   1:L PR[91] R[100]mm/sec CNT100;
   1:  PR[GP1:91,1] = PR[GP1:90,1] + 70.472;
   1:  PR[GP1:91,2] = PR[GP1:90,2] + 15.297;
   1:L PR[91] R[100]mm/sec CNT100;
   1:  PR[GP1:91,1] = PR[GP1:90,1] + 68.185;
   1:  PR[GP1:91,2] = PR[GP1:90,2] + 19.487;
   1:L PR[91] R[100]mm/sec CNT100;
   1:  PR[GP1:91,1] = PR[GP1:90,1] + 65.966;
   1:  PR[GP1:91,2] = PR[GP1:90,2] + 22.379;
   1:L PR[91] R[100]mm/sec CNT100;
   1:  PR[GP1:91,1] = PR[GP1:90,1] + 63.212;
   1:  PR[GP1:91,2] = PR[GP1:90,2] + 24.842;
   1:L PR[91] R[100]mm/sec CNT100;
   1:  PR[GP1:91,1] = PR[GP1:90,1] + 59.563;
   1:  PR[GP1:91,2] = PR[GP1:90,2] + 28.170;
   1:L PR[91] R[100]mm/sec CNT100;
   1:  PR[GP1:91,1] = PR[GP1:90,1] + 56.581;
   1:  PR[GP1:91,2] = PR[GP1:90,2] + 29.968;
   1:L PR[91] R[100]mm/sec CNT100;
   1:  PR[GP1:91,1] = PR[GP1:90,1] + 53.246;
   1:  PR[GP1:91,2] = PR[GP1:90,2] + 31.207;
   1:L PR[91] R[100]mm/sec CNT100;
   1:  PR[GP1:91,1] = PR[GP1:90,1] + 48.490;
   1:  PR[GP1:91,2] = PR[GP1:90,2] + 33.267;
   1:L PR[91] R[100]mm/sec CNT100;
   1:  PR[GP1:91,1] = PR[GP1:90,1] + 45.251;
   1:  PR[GP1:91,2] = PR[GP1:90,2] + 33.819;
   1:L PR[91] R[100]mm/sec CNT100;
   1:  PR[GP1:91,1] = PR[GP1:90,1] + 39.491;
   1:  PR[GP1:91,2] = PR[GP1:90,2] + 34.252;
   1:L PR[91] R[100]mm/sec CNT100;
   1:  PR[GP1:91,1] = PR[GP1:90,1] + 36.457;
   1:  PR[GP1:91,2] = PR[GP1:90,2] + 34.197;
   1:L PR[91] R[100]mm/sec CNT100;
   1:  PR[GP1:91,1] = PR[GP1:90,1] + 33.474;
   1:  PR[GP1:91,2] = PR[GP1:90,2] + 33.576;
   1:L PR[91] R[100]mm/sec CNT100;
   1:  PR[GP1:91,1] = PR[GP1:90,1] + 27.456;
   1:  PR[GP1:91,2] = PR[GP1:90,2] + 32.002;
   1:L PR[91] R[100]mm/sec CNT100;
   1:  PR[GP1:91,1] = PR[GP1:90,1] + 24.948;
   1:  PR[GP1:91,2] = PR[GP1:90,2] + 30.965;
   1:L PR[91] R[100]mm/sec CNT100;
   1:  PR[GP1:91,1] = PR[GP1:90,1] + 22.645;
   1:  PR[GP1:91,2] = PR[GP1:90,2] + 29.460;
   1:L PR[91] R[100]mm/sec CNT100;
   1:  PR[GP1:91,1] = PR[GP1:90,1] + 17.064;
   1:  PR[GP1:91,2] = PR[GP1:90,2] + 25.755;
   1:L PR[91] R[100]mm/sec CNT100;
   1:  PR[GP1:91,1] = PR[GP1:90,1] + 15.344;
   1:  PR[GP1:91,2] = PR[GP1:90,2] + 24.100;
   1:L PR[91] R[100]mm/sec CNT100;
   1:  PR[GP1:91,1] = PR[GP1:90,1] + 13.923;
   1:  PR[GP1:91,2] = PR[GP1:90,2] + 22.102;
   1:L PR[91] R[100]mm/sec CNT100;
   1:  PR[GP1:91,1] = PR[GP1:90,1] + 9.561;
   1:  PR[GP1:91,2] = PR[GP1:90,2] + 16.404;
   1:L PR[91] R[100]mm/sec CNT100;
   1:  PR[GP1:91,1] = PR[GP1:90,1] + 8.670;
   1:  PR[GP1:91,2] = PR[GP1:90,2] + 14.466;
   1:L PR[91] R[100]mm/sec CNT100;
   1:  PR[GP1:91,1] = PR[GP1:90,1] + 6.222;
   1:  PR[GP1:91,2] = PR[GP1:90,2] + 7.080;
   1:L PR[91] R[100]mm/sec CNT100;
   1:  PR[GP1:91,1] = PR[GP1:90,1] + 5.845;
   1:  PR[GP1:91,2] = PR[GP1:90,2] + 5.563;
   1:L PR[91] R[100]mm/sec CNT100;
   1:  PR[GP1:91,1] = PR[GP1:90,1] + 5.869;
   1:  PR[GP1:91,2] = PR[GP1:90,2] + 5.549;
   1:L PR[91] R[100]mm/sec CNT100;
   1:  PR[GP1:91,1] = PR[GP1:90,1] + 5.812;
   1:  PR[GP1:91,2] = PR[GP1:90,2] + 5.029;
   1:L PR[91] R[100]mm/sec CNT100;
   1:  PR[GP1:91,1] = PR[GP1:90,1] + 5.410;
   1:  PR[GP1:91,2] = PR[GP1:90,2] + 4.073;
   1:L PR[91] R[100]mm/sec CNT100;
   1:  PR[GP1:91,1] = PR[GP1:90,1] + 5.006;
   1:  PR[GP1:91,2] = PR[GP1:90,2] + 3.295;
   1:L PR[91] R[100]mm/sec CNT100;
   1:  PR[GP1:91,1] = PR[GP1:90,1] + 4.488;
   1:  PR[GP1:91,2] = PR[GP1:90,2] + 2.358;
   1:L PR[91] R[100]mm/sec CNT100;
   1:  PR[GP1:91,1] = PR[GP1:90,1] + 3.900;
   1:  PR[GP1:91,2] = PR[GP1:90,2] + 1.720;
   1:L PR[91] R[100]mm/sec CNT100;
   1:  PR[GP1:91,1] = PR[GP1:90,1] + 3.010;
   1:  PR[GP1:91,2] = PR[GP1:90,2] + 1.107;
   1:L PR[91] R[100]mm/sec CNT100;
   1:  PR[GP1:91,1] = PR[GP1:90,1] + 2.104;
   1:  PR[GP1:91,2] = PR[GP1:90,2] + 0.771;
   1:L PR[91] R[100]mm/sec CNT100;
   1:  PR[GP1:91,1] = PR[GP1:90,1] + 1.542;
   1:  PR[GP1:91,2] = PR[GP1:90,2] + 0.621;
   1:L PR[91] R[100]mm/sec CNT100;
   1:  PR[GP1:91,1] = PR[GP1:90,1] + 0.324;
   1:  PR[GP1:91,2] = PR[GP1:90,2] + 0.328;
   1:L PR[91] R[100]mm/sec CNT100;
   1:  PR[GP1:91,1] = PR[GP1:90,1] + -0.154;
   1:L PR[91] R[100]mm/sec CNT100;
   1:  ! -- Layer/Ebene 22 -- !;
   1:  PR[91] = PR[90];
   1:  PR[GP1:91,1] = PR[GP1:90,1] + -0.443;
   1:  PR[GP1:91,2] = PR[GP1:90,2] + 0.471;
   1:  PR[GP1:91,3] = PR[GP1:90,3] + 13.725;
   1:L PR[91] R[100]mm/sec CNT100;
   1:  PR[GP1:91,1] = PR[GP1:90,1] + -0.647;
   1:  PR[GP1:91,2] = PR[GP1:90,2] + 0.480;
   1:L PR[91] R[100]mm/sec CNT100;
   1:  PR[GP1:91,1] = PR[GP1:90,1] + -3.627;
   1:  PR[GP1:91,2] = PR[GP1:90,2] + 1.659;
   1:L PR[91] R[100]mm/sec CNT100;
   1:  PR[GP1:91,1] = PR[GP1:90,1] + -3.980;
   1:  PR[GP1:91,2] = PR[GP1:90,2] + 2.296;
   1:L PR[91] R[100]mm/sec CNT100;
   1:  PR[GP1:91,1] = PR[GP1:90,1] + -4.040;
   1:  PR[GP1:91,2] = PR[GP1:90,2] + 2.351;
   1:L PR[91] R[100]mm/sec CNT100;
   1:  PR[GP1:91,1] = PR[GP1:90,1] + -4.473;
   1:  PR[GP1:91,2] = PR[GP1:90,2] + 3.055;
   1:L PR[91] R[100]mm/sec CNT100;
   1:  PR[GP1:91,1] = PR[GP1:90,1] + -5.526;
   1:  PR[GP1:91,2] = PR[GP1:90,2] + 4.999;
   1:L PR[91] R[100]mm/sec CNT100;
   1:  PR[GP1:91,1] = PR[GP1:90,1] + -5.589;
   1:  PR[GP1:91,2] = PR[GP1:90,2] + 5.579;
   1:L PR[91] R[100]mm/sec CNT100;
   1:  PR[GP1:91,1] = PR[GP1:90,1] + -5.827;
   1:  PR[GP1:91,2] = PR[GP1:90,2] + 6.538;
   1:L PR[91] R[100]mm/sec CNT100;
   1:  PR[GP1:91,1] = PR[GP1:90,1] + -8.589;
   1:  PR[GP1:91,2] = PR[GP1:90,2] + 14.871;
   1:L PR[91] R[100]mm/sec CNT100;
   1:  PR[GP1:91,1] = PR[GP1:90,1] + -9.257;
   1:  PR[GP1:91,2] = PR[GP1:90,2] + 16.324;
   1:L PR[91] R[100]mm/sec CNT100;
   1:  PR[GP1:91,1] = PR[GP1:90,1] + -10.196;
   1:  PR[GP1:91,2] = PR[GP1:90,2] + 17.645;
   1:L PR[91] R[100]mm/sec CNT100;
   1:  PR[GP1:91,1] = PR[GP1:90,1] + -15.288;
   1:  PR[GP1:91,2] = PR[GP1:90,2] + 24.311;
   1:L PR[91] R[100]mm/sec CNT100;
   1:  PR[GP1:91,1] = PR[GP1:90,1] + -16.646;
   1:  PR[GP1:91,2] = PR[GP1:90,2] + 25.617;
   1:L PR[91] R[100]mm/sec CNT100;
   1:  PR[GP1:91,1] = PR[GP1:90,1] + -18.262;
   1:  PR[GP1:91,2] = PR[GP1:90,2] + 26.674;
   1:L PR[91] R[100]mm/sec CNT100;
   1:  PR[GP1:91,1] = PR[GP1:90,1] + -24.852;
   1:  PR[GP1:91,2] = PR[GP1:90,2] + 31.045;
   1:L PR[91] R[100]mm/sec CNT100;
   1:  PR[GP1:91,1] = PR[GP1:90,1] + -26.907;
   1:  PR[GP1:91,2] = PR[GP1:90,2] + 31.895;
   1:L PR[91] R[100]mm/sec CNT100;
   1:  PR[GP1:91,1] = PR[GP1:90,1] + -29.156;
   1:  PR[GP1:91,2] = PR[GP1:90,2] + 32.362;
   1:L PR[91] R[100]mm/sec CNT100;
   1:  PR[GP1:91,1] = PR[GP1:90,1] + -36.283;
   1:  PR[GP1:91,2] = PR[GP1:90,2] + 34.208;
   1:L PR[91] R[100]mm/sec CNT100;
   1:  PR[GP1:91,1] = PR[GP1:90,1] + -38.869;
   1:  PR[GP1:91,2] = PR[GP1:90,2] + 34.255;
   1:L PR[91] R[100]mm/sec CNT100;
   1:  PR[GP1:91,1] = PR[GP1:90,1] + -45.366;
   1:  PR[GP1:91,2] = PR[GP1:90,2] + 33.766;
   1:L PR[91] R[100]mm/sec CNT100;
   1:  PR[GP1:91,1] = PR[GP1:90,1] + -48.228;
   1:  PR[GP1:91,2] = PR[GP1:90,2] + 33.279;
   1:L PR[91] R[100]mm/sec CNT100;
   1:  PR[GP1:91,1] = PR[GP1:90,1] + -50.961;
   1:  PR[GP1:91,2] = PR[GP1:90,2] + 32.263;
   1:L PR[91] R[100]mm/sec CNT100;
   1:  PR[GP1:91,1] = PR[GP1:90,1] + -56.550;
   1:  PR[GP1:91,2] = PR[GP1:90,2] + 29.856;
   1:L PR[91] R[100]mm/sec CNT100;
   1:  PR[GP1:91,1] = PR[GP1:90,1] + -59.229;
   1:  PR[GP1:91,2] = PR[GP1:90,2] + 28.240;
   1:L PR[91] R[100]mm/sec CNT100;
   1:  PR[GP1:91,1] = PR[GP1:90,1] + -61.590;
   1:  PR[GP1:91,2] = PR[GP1:90,2] + 26.129;
   1:L PR[91] R[100]mm/sec CNT100;
   1:  PR[GP1:91,1] = PR[GP1:90,1] + -65.832;
   1:  PR[GP1:91,2] = PR[GP1:90,2] + 22.263;
   1:L PR[91] R[100]mm/sec CNT100;
   1:  PR[GP1:91,1] = PR[GP1:90,1] + -67.832;
   1:  PR[GP1:91,2] = PR[GP1:90,2] + 19.657;
   1:L PR[91] R[100]mm/sec CNT100;
   1:  PR[GP1:91,1] = PR[GP1:90,1] + -69.340;
   1:  PR[GP1:91,2] = PR[GP1:90,2] + 16.667;
   1:L PR[91] R[100]mm/sec CNT100;
   1:  PR[GP1:91,1] = PR[GP1:90,1] + -71.966;
   1:  PR[GP1:91,2] = PR[GP1:90,2] + 11.848;
   1:L PR[91] R[100]mm/sec CNT100;
   1:  PR[GP1:91,1] = PR[GP1:90,1] + -72.899;
   1:  PR[GP1:91,2] = PR[GP1:90,2] + 8.606;
   1:L PR[91] R[100]mm/sec CNT100;
   1:  PR[GP1:91,1] = PR[GP1:90,1] + -73.222;
   1:  PR[GP1:91,2] = PR[GP1:90,2] + 5.161;
   1:L PR[91] R[100]mm/sec CNT100;
   1:  PR[GP1:91,1] = PR[GP1:90,1] + -74.099;
   1:  PR[GP1:91,2] = PR[GP1:90,2] + -0.094;
   1:L PR[91] R[100]mm/sec CNT100;
   1:  PR[GP1:91,1] = PR[GP1:90,1] + -73.772;
   1:  PR[GP1:91,2] = PR[GP1:90,2] + -3.582;
   1:L PR[91] R[100]mm/sec CNT100;
   1:  PR[GP1:91,1] = PR[GP1:90,1] + -72.906;
   1:  PR[GP1:91,2] = PR[GP1:90,2] + -8.729;
   1:L PR[91] R[100]mm/sec CNT100;
   1:  PR[GP1:91,1] = PR[GP1:90,1] + -71.963;
   1:  PR[GP1:91,2] = PR[GP1:90,2] + -12.001;
   1:L PR[91] R[100]mm/sec CNT100;
   1:  PR[GP1:91,1] = PR[GP1:90,1] + -70.418;
   1:  PR[GP1:91,2] = PR[GP1:90,2] + -15.062;
   1:L PR[91] R[100]mm/sec CNT100;
   1:  PR[GP1:91,1] = PR[GP1:90,1] + -67.838;
   1:  PR[GP1:91,2] = PR[GP1:90,2] + -19.793;
   1:L PR[91] R[100]mm/sec CNT100;
   1:  PR[GP1:91,1] = PR[GP1:90,1] + -65.834;
   1:  PR[GP1:91,2] = PR[GP1:90,2] + -22.405;
   1:L PR[91] R[100]mm/sec CNT100;
   1:  PR[GP1:91,1] = PR[GP1:90,1] + -63.343;
   1:  PR[GP1:91,2] = PR[GP1:90,2] + -24.632;
   1:L PR[91] R[100]mm/sec CNT100;
   1:  PR[GP1:91,1] = PR[GP1:90,1] + -59.227;
   1:  PR[GP1:91,2] = PR[GP1:90,2] + -28.385;
   1:L PR[91] R[100]mm/sec CNT100;
   1:  PR[GP1:91,1] = PR[GP1:90,1] + -56.563;
   1:  PR[GP1:91,2] = PR[GP1:90,2] + -29.992;
   1:L PR[91] R[100]mm/sec CNT100;
   1:  PR[GP1:91,1] = PR[GP1:90,1] + -53.577;
   1:  PR[GP1:91,2] = PR[GP1:90,2] + -31.101;
   1:L PR[91] R[100]mm/sec CNT100;
   1:  PR[GP1:91,1] = PR[GP1:90,1] + -48.212;
   1:  PR[GP1:91,2] = PR[GP1:90,2] + -33.425;
   1:L PR[91] R[100]mm/sec CNT100;
   1:  PR[GP1:91,1] = PR[GP1:90,1] + -45.366;
   1:  PR[GP1:91,2] = PR[GP1:90,2] + -33.910;
   1:L PR[91] R[100]mm/sec CNT100;
   1:  PR[GP1:91,1] = PR[GP1:90,1] + -38.869;
   1:  PR[GP1:91,2] = PR[GP1:90,2] + -34.399;
   1:L PR[91] R[100]mm/sec CNT100;
   1:  PR[GP1:91,1] = PR[GP1:90,1] + -36.268;
   1:  PR[GP1:91,2] = PR[GP1:90,2] + -34.352;
   1:L PR[91] R[100]mm/sec CNT100;
   1:  PR[GP1:91,1] = PR[GP1:90,1] + -33.709;
   1:  PR[GP1:91,2] = PR[GP1:90,2] + -33.819;
   1:L PR[91] R[100]mm/sec CNT100;
   1:  PR[GP1:91,1] = PR[GP1:90,1] + -26.921;
   1:  PR[GP1:91,2] = PR[GP1:90,2] + -32.044;
   1:L PR[91] R[100]mm/sec CNT100;
   1:  PR[GP1:91,1] = PR[GP1:90,1] + -24.850;
   1:  PR[GP1:91,2] = PR[GP1:90,2] + -31.188;
   1:L PR[91] R[100]mm/sec CNT100;
   1:  PR[GP1:91,1] = PR[GP1:90,1] + -22.942;
   1:  PR[GP1:91,2] = PR[GP1:90,2] + -29.941;
   1:L PR[91] R[100]mm/sec CNT100;
   1:  PR[GP1:91,1] = PR[GP1:90,1] + -16.647;
   1:  PR[GP1:91,2] = PR[GP1:90,2] + -25.762;
   1:L PR[91] R[100]mm/sec CNT100;
   1:  PR[GP1:91,1] = PR[GP1:90,1] + -15.296;
   1:  PR[GP1:91,2] = PR[GP1:90,2] + -24.463;
   1:L PR[91] R[100]mm/sec CNT100;
   1:  PR[GP1:91,1] = PR[GP1:90,1] + -14.172;
   1:  PR[GP1:91,2] = PR[GP1:90,2] + -22.882;
   1:L PR[91] R[100]mm/sec CNT100;
   1:  PR[GP1:91,1] = PR[GP1:90,1] + -9.252;
   1:  PR[GP1:91,2] = PR[GP1:90,2] + -16.458;
   1:L PR[91] R[100]mm/sec CNT100;
   1:  PR[GP1:91,1] = PR[GP1:90,1] + -8.589;
   1:  PR[GP1:91,2] = PR[GP1:90,2] + -15.015;
   1:L PR[91] R[100]mm/sec CNT100;
   1:  PR[GP1:91,1] = PR[GP1:90,1] + -5.828;
   1:  PR[GP1:91,2] = PR[GP1:90,2] + -6.684;
   1:L PR[91] R[100]mm/sec CNT100;
   1:  PR[GP1:91,1] = PR[GP1:90,1] + -5.587;
   1:  PR[GP1:91,2] = PR[GP1:90,2] + -5.718;
   1:L PR[91] R[100]mm/sec CNT100;
   1:  PR[GP1:91,1] = PR[GP1:90,1] + -5.590;
   1:  PR[GP1:91,2] = PR[GP1:90,2] + -5.716;
   1:L PR[91] R[100]mm/sec CNT100;
   1:  PR[GP1:91,1] = PR[GP1:90,1] + -5.530;
   1:  PR[GP1:91,2] = PR[GP1:90,2] + -5.173;
   1:L PR[91] R[100]mm/sec CNT100;
   1:  PR[GP1:91,1] = PR[GP1:90,1] + -4.941;
   1:  PR[GP1:91,2] = PR[GP1:90,2] + -3.769;
   1:L PR[91] R[100]mm/sec CNT100;
   1:  PR[GP1:91,1] = PR[GP1:90,1] + -4.300;
   1:  PR[GP1:91,2] = PR[GP1:90,2] + -2.578;
   1:L PR[91] R[100]mm/sec CNT100;
   1:  PR[GP1:91,1] = PR[GP1:90,1] + -3.647;
   1:  PR[GP1:91,2] = PR[GP1:90,2] + -1.869;
   1:L PR[91] R[100]mm/sec CNT100;
   1:  PR[GP1:91,1] = PR[GP1:90,1] + -2.659;
   1:  PR[GP1:91,2] = PR[GP1:90,2] + -1.188;
   1:L PR[91] R[100]mm/sec CNT100;
   1:  PR[GP1:91,1] = PR[GP1:90,1] + -2.064;
   1:  PR[GP1:91,2] = PR[GP1:90,2] + -0.967;
   1:L PR[91] R[100]mm/sec CNT100;
   1:  PR[GP1:91,1] = PR[GP1:90,1] + -1.705;
   1:  PR[GP1:91,2] = PR[GP1:90,2] + -0.872;
   1:L PR[91] R[100]mm/sec CNT100;
   1:  PR[GP1:91,1] = PR[GP1:90,1] + -0.043;
   1:  PR[GP1:91,2] = PR[GP1:90,2] + -0.472;
   1:L PR[91] R[100]mm/sec CNT100;
   1:  PR[GP1:91,1] = PR[GP1:90,1] + 0.299;
   1:L PR[91] R[100]mm/sec CNT100;
   1:  PR[GP1:91,1] = PR[GP1:90,1] + 0.657;
   1:  PR[GP1:91,2] = PR[GP1:90,2] + -0.615;
   1:L PR[91] R[100]mm/sec CNT100;
   1:  PR[GP1:91,1] = PR[GP1:90,1] + 0.860;
   1:  PR[GP1:91,2] = PR[GP1:90,2] + -0.623;
   1:L PR[91] R[100]mm/sec CNT100;
   1:  PR[GP1:91,1] = PR[GP1:90,1] + 3.841;
   1:  PR[GP1:91,2] = PR[GP1:90,2] + -1.803;
   1:L PR[91] R[100]mm/sec CNT100;
   1:  PR[GP1:91,1] = PR[GP1:90,1] + 4.193;
   1:  PR[GP1:91,2] = PR[GP1:90,2] + -2.440;
   1:L PR[91] R[100]mm/sec CNT100;
   1:  PR[GP1:91,1] = PR[GP1:90,1] + 4.254;
   1:  PR[GP1:91,2] = PR[GP1:90,2] + -2.495;
   1:L PR[91] R[100]mm/sec CNT100;
   1:  PR[GP1:91,1] = PR[GP1:90,1] + 4.687;
   1:  PR[GP1:91,2] = PR[GP1:90,2] + -3.199;
   1:L PR[91] R[100]mm/sec CNT100;
   1:  PR[GP1:91,1] = PR[GP1:90,1] + 5.739;
   1:  PR[GP1:91,2] = PR[GP1:90,2] + -5.143;
   1:L PR[91] R[100]mm/sec CNT100;
   1:  PR[GP1:91,1] = PR[GP1:90,1] + 5.802;
   1:  PR[GP1:91,2] = PR[GP1:90,2] + -5.723;
   1:L PR[91] R[100]mm/sec CNT100;
   1:  PR[GP1:91,1] = PR[GP1:90,1] + 6.040;
   1:  PR[GP1:91,2] = PR[GP1:90,2] + -6.685;
   1:L PR[91] R[100]mm/sec CNT100;
   1:  PR[GP1:91,1] = PR[GP1:90,1] + 8.801;
   1:  PR[GP1:91,2] = PR[GP1:90,2] + -15.012;
   1:L PR[91] R[100]mm/sec CNT100;
   1:  PR[GP1:91,1] = PR[GP1:90,1] + 9.469;
   1:  PR[GP1:91,2] = PR[GP1:90,2] + -16.464;
   1:L PR[91] R[100]mm/sec CNT100;
   1:  PR[GP1:91,1] = PR[GP1:90,1] + 10.408;
   1:  PR[GP1:91,2] = PR[GP1:90,2] + -17.786;
   1:L PR[91] R[100]mm/sec CNT100;
   1:  PR[GP1:91,1] = PR[GP1:90,1] + 15.500;
   1:  PR[GP1:91,2] = PR[GP1:90,2] + -24.455;
   1:L PR[91] R[100]mm/sec CNT100;
   1:  PR[GP1:91,1] = PR[GP1:90,1] + 16.857;
   1:  PR[GP1:91,2] = PR[GP1:90,2] + -25.760;
   1:L PR[91] R[100]mm/sec CNT100;
   1:  PR[GP1:91,1] = PR[GP1:90,1] + 18.474;
   1:  PR[GP1:91,2] = PR[GP1:90,2] + -26.817;
   1:L PR[91] R[100]mm/sec CNT100;
   1:  PR[GP1:91,1] = PR[GP1:90,1] + 25.063;
   1:  PR[GP1:91,2] = PR[GP1:90,2] + -31.188;
   1:L PR[91] R[100]mm/sec CNT100;
   1:  PR[GP1:91,1] = PR[GP1:90,1] + 27.119;
   1:  PR[GP1:91,2] = PR[GP1:90,2] + -32.038;
   1:L PR[91] R[100]mm/sec CNT100;
   1:  PR[GP1:91,1] = PR[GP1:90,1] + 29.367;
   1:  PR[GP1:91,2] = PR[GP1:90,2] + -32.506;
   1:L PR[91] R[100]mm/sec CNT100;
   1:  PR[GP1:91,1] = PR[GP1:90,1] + 36.495;
   1:  PR[GP1:91,2] = PR[GP1:90,2] + -34.352;
   1:L PR[91] R[100]mm/sec CNT100;
   1:  PR[GP1:91,1] = PR[GP1:90,1] + 39.081;
   1:  PR[GP1:91,2] = PR[GP1:90,2] + -34.399;
   1:L PR[91] R[100]mm/sec CNT100;
   1:  PR[GP1:91,1] = PR[GP1:90,1] + 45.579;
   1:  PR[GP1:91,2] = PR[GP1:90,2] + -33.910;
   1:L PR[91] R[100]mm/sec CNT100;
   1:  PR[GP1:91,1] = PR[GP1:90,1] + 48.441;
   1:  PR[GP1:91,2] = PR[GP1:90,2] + -33.423;
   1:L PR[91] R[100]mm/sec CNT100;
   1:  PR[GP1:91,1] = PR[GP1:90,1] + 51.174;
   1:  PR[GP1:91,2] = PR[GP1:90,2] + -32.407;
   1:L PR[91] R[100]mm/sec CNT100;
   1:  PR[GP1:91,1] = PR[GP1:90,1] + 56.763;
   1:  PR[GP1:91,2] = PR[GP1:90,2] + -30.000;
   1:L PR[91] R[100]mm/sec CNT100;
   1:  PR[GP1:91,1] = PR[GP1:90,1] + 59.442;
   1:  PR[GP1:91,2] = PR[GP1:90,2] + -28.385;
   1:L PR[91] R[100]mm/sec CNT100;
   1:  PR[GP1:91,1] = PR[GP1:90,1] + 61.803;
   1:  PR[GP1:91,2] = PR[GP1:90,2] + -26.274;
   1:L PR[91] R[100]mm/sec CNT100;
   1:  PR[GP1:91,1] = PR[GP1:90,1] + 66.045;
   1:  PR[GP1:91,2] = PR[GP1:90,2] + -22.407;
   1:L PR[91] R[100]mm/sec CNT100;
   1:  PR[GP1:91,1] = PR[GP1:90,1] + 68.045;
   1:  PR[GP1:91,2] = PR[GP1:90,2] + -19.800;
   1:L PR[91] R[100]mm/sec CNT100;
   1:  PR[GP1:91,1] = PR[GP1:90,1] + 69.553;
   1:  PR[GP1:91,2] = PR[GP1:90,2] + -16.810;
   1:L PR[91] R[100]mm/sec CNT100;
   1:  PR[GP1:91,1] = PR[GP1:90,1] + 72.179;
   1:  PR[GP1:91,2] = PR[GP1:90,2] + -11.994;
   1:L PR[91] R[100]mm/sec CNT100;
   1:  PR[GP1:91,1] = PR[GP1:90,1] + 73.113;
   1:  PR[GP1:91,2] = PR[GP1:90,2] + -8.752;
   1:L PR[91] R[100]mm/sec CNT100;
   1:  PR[GP1:91,1] = PR[GP1:90,1] + 73.436;
   1:  PR[GP1:91,2] = PR[GP1:90,2] + -5.307;
   1:L PR[91] R[100]mm/sec CNT100;
   1:  PR[GP1:91,1] = PR[GP1:90,1] + 74.312;
   1:  PR[GP1:91,2] = PR[GP1:90,2] + -0.050;
   1:L PR[91] R[100]mm/sec CNT100;
   1:  PR[GP1:91,1] = PR[GP1:90,1] + 73.985;
   1:  PR[GP1:91,2] = PR[GP1:90,2] + 3.438;
   1:L PR[91] R[100]mm/sec CNT100;
   1:  PR[GP1:91,1] = PR[GP1:90,1] + 73.119;
   1:  PR[GP1:91,2] = PR[GP1:90,2] + 8.587;
   1:L PR[91] R[100]mm/sec CNT100;
   1:  PR[GP1:91,1] = PR[GP1:90,1] + 72.176;
   1:  PR[GP1:91,2] = PR[GP1:90,2] + 11.859;
   1:L PR[91] R[100]mm/sec CNT100;
   1:  PR[GP1:91,1] = PR[GP1:90,1] + 70.632;
   1:  PR[GP1:91,2] = PR[GP1:90,2] + 14.920;
   1:L PR[91] R[100]mm/sec CNT100;
   1:  PR[GP1:91,1] = PR[GP1:90,1] + 68.051;
   1:  PR[GP1:91,2] = PR[GP1:90,2] + 19.648;
   1:L PR[91] R[100]mm/sec CNT100;
   1:  PR[GP1:91,1] = PR[GP1:90,1] + 66.047;
   1:  PR[GP1:91,2] = PR[GP1:90,2] + 22.260;
   1:L PR[91] R[100]mm/sec CNT100;
   1:  PR[GP1:91,1] = PR[GP1:90,1] + 63.556;
   1:  PR[GP1:91,2] = PR[GP1:90,2] + 24.488;
   1:L PR[91] R[100]mm/sec CNT100;
   1:  PR[GP1:91,1] = PR[GP1:90,1] + 59.439;
   1:  PR[GP1:91,2] = PR[GP1:90,2] + 28.242;
   1:L PR[91] R[100]mm/sec CNT100;
   1:  PR[GP1:91,1] = PR[GP1:90,1] + 56.776;
   1:  PR[GP1:91,2] = PR[GP1:90,2] + 29.848;
   1:L PR[91] R[100]mm/sec CNT100;
   1:  PR[GP1:91,1] = PR[GP1:90,1] + 53.790;
   1:  PR[GP1:91,2] = PR[GP1:90,2] + 30.958;
   1:L PR[91] R[100]mm/sec CNT100;
   1:  PR[GP1:91,1] = PR[GP1:90,1] + 48.425;
   1:  PR[GP1:91,2] = PR[GP1:90,2] + 33.281;
   1:L PR[91] R[100]mm/sec CNT100;
   1:  PR[GP1:91,1] = PR[GP1:90,1] + 45.579;
   1:  PR[GP1:91,2] = PR[GP1:90,2] + 33.766;
   1:L PR[91] R[100]mm/sec CNT100;
   1:  PR[GP1:91,1] = PR[GP1:90,1] + 39.081;
   1:  PR[GP1:91,2] = PR[GP1:90,2] + 34.255;
   1:L PR[91] R[100]mm/sec CNT100;
   1:  PR[GP1:91,1] = PR[GP1:90,1] + 36.480;
   1:  PR[GP1:91,2] = PR[GP1:90,2] + 34.208;
   1:L PR[91] R[100]mm/sec CNT100;
   1:  PR[GP1:91,1] = PR[GP1:90,1] + 33.921;
   1:  PR[GP1:91,2] = PR[GP1:90,2] + 33.675;
   1:L PR[91] R[100]mm/sec CNT100;
   1:  PR[GP1:91,1] = PR[GP1:90,1] + 27.133;
   1:  PR[GP1:91,2] = PR[GP1:90,2] + 31.900;
   1:L PR[91] R[100]mm/sec CNT100;
   1:  PR[GP1:91,1] = PR[GP1:90,1] + 25.062;
   1:  PR[GP1:91,2] = PR[GP1:90,2] + 31.043;
   1:L PR[91] R[100]mm/sec CNT100;
   1:  PR[GP1:91,1] = PR[GP1:90,1] + 23.153;
   1:  PR[GP1:91,2] = PR[GP1:90,2] + 29.796;
   1:L PR[91] R[100]mm/sec CNT100;
   1:  PR[GP1:91,1] = PR[GP1:90,1] + 16.859;
   1:  PR[GP1:91,2] = PR[GP1:90,2] + 25.618;
   1:L PR[91] R[100]mm/sec CNT100;
   1:  PR[GP1:91,1] = PR[GP1:90,1] + 15.508;
   1:  PR[GP1:91,2] = PR[GP1:90,2] + 24.318;
   1:L PR[91] R[100]mm/sec CNT100;
   1:  PR[GP1:91,1] = PR[GP1:90,1] + 14.384;
   1:  PR[GP1:91,2] = PR[GP1:90,2] + 22.737;
   1:L PR[91] R[100]mm/sec CNT100;
   1:  PR[GP1:91,1] = PR[GP1:90,1] + 9.464;
   1:  PR[GP1:91,2] = PR[GP1:90,2] + 16.311;
   1:L PR[91] R[100]mm/sec CNT100;
   1:  PR[GP1:91,1] = PR[GP1:90,1] + 8.801;
   1:  PR[GP1:91,2] = PR[GP1:90,2] + 14.868;
   1:L PR[91] R[100]mm/sec CNT100;
   1:  PR[GP1:91,1] = PR[GP1:90,1] + 6.040;
   1:  PR[GP1:91,2] = PR[GP1:90,2] + 6.538;
   1:L PR[91] R[100]mm/sec CNT100;
   1:  PR[GP1:91,1] = PR[GP1:90,1] + 5.800;
   1:  PR[GP1:91,2] = PR[GP1:90,2] + 5.575;
   1:L PR[91] R[100]mm/sec CNT100;
   1:  PR[GP1:91,1] = PR[GP1:90,1] + 5.803;
   1:  PR[GP1:91,2] = PR[GP1:90,2] + 5.574;
   1:L PR[91] R[100]mm/sec CNT100;
   1:  PR[GP1:91,1] = PR[GP1:90,1] + 5.743;
   1:  PR[GP1:91,2] = PR[GP1:90,2] + 5.029;
   1:L PR[91] R[100]mm/sec CNT100;
   1:  PR[GP1:91,1] = PR[GP1:90,1] + 5.155;
   1:  PR[GP1:91,2] = PR[GP1:90,2] + 3.627;
   1:L PR[91] R[100]mm/sec CNT100;
   1:  PR[GP1:91,1] = PR[GP1:90,1] + 4.513;
   1:  PR[GP1:91,2] = PR[GP1:90,2] + 2.434;
   1:L PR[91] R[100]mm/sec CNT100;
   1:  PR[GP1:91,1] = PR[GP1:90,1] + 3.860;
   1:  PR[GP1:91,2] = PR[GP1:90,2] + 1.725;
   1:L PR[91] R[100]mm/sec CNT100;
   1:  PR[GP1:91,1] = PR[GP1:90,1] + 2.873;
   1:  PR[GP1:91,2] = PR[GP1:90,2] + 1.044;
   1:L PR[91] R[100]mm/sec CNT100;
   1:  PR[GP1:91,1] = PR[GP1:90,1] + 2.277;
   1:  PR[GP1:91,2] = PR[GP1:90,2] + 0.823;
   1:L PR[91] R[100]mm/sec CNT100;
   1:  PR[GP1:91,1] = PR[GP1:90,1] + 1.917;
   1:  PR[GP1:91,2] = PR[GP1:90,2] + 0.727;
   1:L PR[91] R[100]mm/sec CNT100;
   1:  PR[GP1:91,1] = PR[GP1:90,1] + 0.256;
   1:  PR[GP1:91,2] = PR[GP1:90,2] + 0.328;
   1:L PR[91] R[100]mm/sec CNT100;
   1:  PR[GP1:91,1] = PR[GP1:90,1] + -0.086;
   1:L PR[91] R[100]mm/sec CNT100;
   1:  ! -- Layer/Ebene 23 -- !;
   1:  PR[91] = PR[90];
   1:  PR[GP1:91,1] = PR[GP1:90,1] + -0.300;
   1:  PR[GP1:91,2] = PR[GP1:90,2] + 0.360;
   1:  PR[GP1:91,3] = PR[GP1:90,3] + 14.335;
   1:L PR[91] R[100]mm/sec CNT100;
   1:  PR[GP1:91,1] = PR[GP1:90,1] + -3.582;
   1:  PR[GP1:91,2] = PR[GP1:90,2] + 1.659;
   1:L PR[91] R[100]mm/sec CNT100;
   1:  PR[GP1:91,1] = PR[GP1:90,1] + -3.779;
   1:  PR[GP1:91,2] = PR[GP1:90,2] + 2.014;
   1:L PR[91] R[100]mm/sec CNT100;
   1:  PR[GP1:91,1] = PR[GP1:90,1] + -3.847;
   1:  PR[GP1:91,2] = PR[GP1:90,2] + 2.076;
   1:L PR[91] R[100]mm/sec CNT100;
   1:  PR[GP1:91,1] = PR[GP1:90,1] + -4.082;
   1:  PR[GP1:91,2] = PR[GP1:90,2] + 2.458;
   1:L PR[91] R[100]mm/sec CNT100;
   1:  PR[GP1:91,1] = PR[GP1:90,1] + -5.458;
   1:  PR[GP1:91,2] = PR[GP1:90,2] + 4.999;
   1:L PR[91] R[100]mm/sec CNT100;
   1:  PR[GP1:91,1] = PR[GP1:90,1] + -5.506;
   1:  PR[GP1:91,2] = PR[GP1:90,2] + 5.437;
   1:L PR[91] R[100]mm/sec CNT100;
   1:  PR[GP1:91,1] = PR[GP1:90,1] + -5.645;
   1:  PR[GP1:91,2] = PR[GP1:90,2] + 5.996;
   1:L PR[91] R[100]mm/sec CNT100;
   1:  PR[GP1:91,1] = PR[GP1:90,1] + -8.719;
   1:  PR[GP1:91,2] = PR[GP1:90,2] + 15.274;
   1:L PR[91] R[100]mm/sec CNT100;
   1:  PR[GP1:91,1] = PR[GP1:90,1] + -9.159;
   1:  PR[GP1:91,2] = PR[GP1:90,2] + 16.231;
   1:L PR[91] R[100]mm/sec CNT100;
   1:  PR[GP1:91,1] = PR[GP1:90,1] + -9.783;
   1:  PR[GP1:91,2] = PR[GP1:90,2] + 17.108;
   1:L PR[91] R[100]mm/sec CNT100;
   1:  PR[GP1:91,1] = PR[GP1:90,1] + -15.452;
   1:  PR[GP1:91,2] = PR[GP1:90,2] + 24.529;
   1:L PR[91] R[100]mm/sec CNT100;
   1:  PR[GP1:91,1] = PR[GP1:90,1] + -16.442;
   1:  PR[GP1:91,2] = PR[GP1:90,2] + 25.481;
   1:L PR[91] R[100]mm/sec CNT100;
   1:  PR[GP1:91,1] = PR[GP1:90,1] + -24.965;
   1:  PR[GP1:91,2] = PR[GP1:90,2] + 31.123;
   1:L PR[91] R[100]mm/sec CNT100;
   1:  PR[GP1:91,1] = PR[GP1:90,1] + -26.584;
   1:  PR[GP1:91,2] = PR[GP1:90,2] + 31.792;
   1:L PR[91] R[100]mm/sec CNT100;
   1:  PR[GP1:91,1] = PR[GP1:90,1] + -28.371;
   1:  PR[GP1:91,2] = PR[GP1:90,2] + 32.164;
   1:L PR[91] R[100]mm/sec CNT100;
   1:  PR[GP1:91,1] = PR[GP1:90,1] + -36.306;
   1:  PR[GP1:91,2] = PR[GP1:90,2] + 34.219;
   1:L PR[91] R[100]mm/sec CNT100;
   1:  PR[GP1:91,1] = PR[GP1:90,1] + -38.459;
   1:  PR[GP1:91,2] = PR[GP1:90,2] + 34.258;
   1:L PR[91] R[100]mm/sec CNT100;
   1:  PR[GP1:91,1] = PR[GP1:90,1] + -45.694;
   1:  PR[GP1:91,2] = PR[GP1:90,2] + 33.714;
   1:L PR[91] R[100]mm/sec CNT100;
   1:  PR[GP1:91,1] = PR[GP1:90,1] + -48.163;
   1:  PR[GP1:91,2] = PR[GP1:90,2] + 33.293;
   1:L PR[91] R[100]mm/sec CNT100;
   1:  PR[GP1:91,1] = PR[GP1:90,1] + -50.522;
   1:  PR[GP1:91,2] = PR[GP1:90,2] + 32.417;
   1:L PR[91] R[100]mm/sec CNT100;
   1:  PR[GP1:91,1] = PR[GP1:90,1] + -56.745;
   1:  PR[GP1:91,2] = PR[GP1:90,2] + 29.736;
   1:L PR[91] R[100]mm/sec CNT100;
   1:  PR[GP1:91,1] = PR[GP1:90,1] + -59.106;
   1:  PR[GP1:91,2] = PR[GP1:90,2] + 28.312;
   1:L PR[91] R[100]mm/sec CNT100;
   1:  PR[GP1:91,1] = PR[GP1:90,1] + -61.189;
   1:  PR[GP1:91,2] = PR[GP1:90,2] + 26.450;
   1:L PR[91] R[100]mm/sec CNT100;
   1:  PR[GP1:91,1] = PR[GP1:90,1] + -65.913;
   1:  PR[GP1:91,2] = PR[GP1:90,2] + 22.144;
   1:L PR[91] R[100]mm/sec CNT100;
   1:  PR[GP1:91,1] = PR[GP1:90,1] + -67.698;
   1:  PR[GP1:91,2] = PR[GP1:90,2] + 19.818;
   1:L PR[91] R[100]mm/sec CNT100;
   1:  PR[GP1:91,1] = PR[GP1:90,1] + -69.047;
   1:  PR[GP1:91,2] = PR[GP1:90,2] + 17.144;
   1:L PR[91] R[100]mm/sec CNT100;
   1:  PR[GP1:91,1] = PR[GP1:90,1] + -71.971;
   1:  PR[GP1:91,2] = PR[GP1:90,2] + 11.776;
   1:L PR[91] R[100]mm/sec CNT100;
   1:  PR[GP1:91,1] = PR[GP1:90,1] + -72.810;
   1:  PR[GP1:91,2] = PR[GP1:90,2] + 8.863;
   1:L PR[91] R[100]mm/sec CNT100;
   1:  PR[GP1:91,1] = PR[GP1:90,1] + -73.101;
   1:  PR[GP1:91,2] = PR[GP1:90,2] + 5.758;
   1:L PR[91] R[100]mm/sec CNT100;
   1:  PR[GP1:91,1] = PR[GP1:90,1] + -74.078;
   1:  PR[GP1:91,2] = PR[GP1:90,2] + -0.094;
   1:L PR[91] R[100]mm/sec CNT100;
   1:  PR[GP1:91,1] = PR[GP1:90,1] + -73.781;
   1:  PR[GP1:91,2] = PR[GP1:90,2] + -3.254;
   1:L PR[91] R[100]mm/sec CNT100;
   1:  PR[GP1:91,1] = PR[GP1:90,1] + -72.816;
   1:  PR[GP1:91,2] = PR[GP1:90,2] + -8.986;
   1:L PR[91] R[100]mm/sec CNT100;
   1:  PR[GP1:91,1] = PR[GP1:90,1] + -71.969;
   1:  PR[GP1:91,2] = PR[GP1:90,2] + -11.929;
   1:L PR[91] R[100]mm/sec CNT100;
   1:  PR[GP1:91,1] = PR[GP1:90,1] + -70.578;
   1:  PR[GP1:91,2] = PR[GP1:90,2] + -14.686;
   1:L PR[91] R[100]mm/sec CNT100;
   1:  PR[GP1:91,1] = PR[GP1:90,1] + -67.704;
   1:  PR[GP1:91,2] = PR[GP1:90,2] + -19.954;
   1:L PR[91] R[100]mm/sec CNT100;
   1:  PR[GP1:91,1] = PR[GP1:90,1] + -65.915;
   1:  PR[GP1:91,2] = PR[GP1:90,2] + -22.286;
   1:L PR[91] R[100]mm/sec CNT100;
   1:  PR[GP1:91,1] = PR[GP1:90,1] + -63.687;
   1:  PR[GP1:91,2] = PR[GP1:90,2] + -24.278;
   1:L PR[91] R[100]mm/sec CNT100;
   1:  PR[GP1:91,1] = PR[GP1:90,1] + -59.103;
   1:  PR[GP1:91,2] = PR[GP1:90,2] + -28.458;
   1:L PR[91] R[100]mm/sec CNT100;
   1:  PR[GP1:91,1] = PR[GP1:90,1] + -56.758;
   1:  PR[GP1:91,2] = PR[GP1:90,2] + -29.872;
   1:L PR[91] R[100]mm/sec CNT100;
   1:  PR[GP1:91,1] = PR[GP1:90,1] + -54.121;
   1:  PR[GP1:91,2] = PR[GP1:90,2] + -30.851;
   1:L PR[91] R[100]mm/sec CNT100;
   1:  PR[GP1:91,1] = PR[GP1:90,1] + -48.147;
   1:  PR[GP1:91,2] = PR[GP1:90,2] + -33.440;
   1:L PR[91] R[100]mm/sec CNT100;
   1:  PR[GP1:91,1] = PR[GP1:90,1] + -45.694;
   1:  PR[GP1:91,2] = PR[GP1:90,2] + -33.858;
   1:L PR[91] R[100]mm/sec CNT100;
   1:  PR[GP1:91,1] = PR[GP1:90,1] + -38.459;
   1:  PR[GP1:91,2] = PR[GP1:90,2] + -34.402;
   1:L PR[91] R[100]mm/sec CNT100;
   1:  PR[GP1:91,1] = PR[GP1:90,1] + -36.291;
   1:  PR[GP1:91,2] = PR[GP1:90,2] + -34.363;
   1:L PR[91] R[100]mm/sec CNT100;
   1:  PR[GP1:91,1] = PR[GP1:90,1] + -34.156;
   1:  PR[GP1:91,2] = PR[GP1:90,2] + -33.918;
   1:L PR[91] R[100]mm/sec CNT100;
   1:  PR[GP1:91,1] = PR[GP1:90,1] + -26.598;
   1:  PR[GP1:91,2] = PR[GP1:90,2] + -31.942;
   1:L PR[91] R[100]mm/sec CNT100;
   1:  PR[GP1:91,1] = PR[GP1:90,1] + -24.963;
   1:  PR[GP1:91,2] = PR[GP1:90,2] + -31.266;
   1:L PR[91] R[100]mm/sec CNT100;
   1:  PR[GP1:91,1] = PR[GP1:90,1] + -23.451;
   1:  PR[GP1:91,2] = PR[GP1:90,2] + -30.277;
   1:L PR[91] R[100]mm/sec CNT100;
   1:  PR[GP1:91,1] = PR[GP1:90,1] + -16.442;
   1:  PR[GP1:91,2] = PR[GP1:90,2] + -25.625;
   1:L PR[91] R[100]mm/sec CNT100;
   1:  PR[GP1:91,1] = PR[GP1:90,1] + -15.460;
   1:  PR[GP1:91,2] = PR[GP1:90,2] + -24.680;
   1:L PR[91] R[100]mm/sec CNT100;
   1:  PR[GP1:91,1] = PR[GP1:90,1] + -14.632;
   1:  PR[GP1:91,2] = PR[GP1:90,2] + -23.516;
   1:L PR[91] R[100]mm/sec CNT100;
   1:  PR[GP1:91,1] = PR[GP1:90,1] + -9.155;
   1:  PR[GP1:91,2] = PR[GP1:90,2] + -16.365;
   1:L PR[91] R[100]mm/sec CNT100;
   1:  PR[GP1:91,1] = PR[GP1:90,1] + -8.719;
   1:  PR[GP1:91,2] = PR[GP1:90,2] + -15.418;
   1:L PR[91] R[100]mm/sec CNT100;
   1:  PR[GP1:91,1] = PR[GP1:90,1] + -5.646;
   1:  PR[GP1:91,2] = PR[GP1:90,2] + -6.142;
   1:L PR[91] R[100]mm/sec CNT100;
   1:  PR[GP1:91,1] = PR[GP1:90,1] + -5.508;
   1:  PR[GP1:91,2] = PR[GP1:90,2] + -5.589;
   1:L PR[91] R[100]mm/sec CNT100;
   1:  PR[GP1:91,1] = PR[GP1:90,1] + -5.462;
   1:  PR[GP1:91,2] = PR[GP1:90,2] + -5.173;
   1:L PR[91] R[100]mm/sec CNT100;
   1:  PR[GP1:91,1] = PR[GP1:90,1] + -4.687;
   1:  PR[GP1:91,2] = PR[GP1:90,2] + -3.328;
   1:L PR[91] R[100]mm/sec CNT100;
   1:  PR[GP1:91,1] = PR[GP1:90,1] + -4.323;
   1:  PR[GP1:91,2] = PR[GP1:90,2] + -2.650;
   1:L PR[91] R[100]mm/sec CNT100;
   1:  PR[GP1:91,1] = PR[GP1:90,1] + -3.607;
   1:  PR[GP1:91,2] = PR[GP1:90,2] + -1.874;
   1:L PR[91] R[100]mm/sec CNT100;
   1:  PR[GP1:91,1] = PR[GP1:90,1] + -2.512;
   1:  PR[GP1:91,2] = PR[GP1:90,2] + -1.119;
   1:L PR[91] R[100]mm/sec CNT100;
   1:  PR[GP1:91,1] = PR[GP1:90,1] + -2.098;
   1:  PR[GP1:91,2] = PR[GP1:90,2] + -0.982;
   1:L PR[91] R[100]mm/sec CNT100;
   1:  PR[GP1:91,1] = PR[GP1:90,1] + 0.106;
   1:  PR[GP1:91,2] = PR[GP1:90,2] + -0.452;
   1:L PR[91] R[100]mm/sec CNT100;
   1:  PR[GP1:91,1] = PR[GP1:90,1] + 0.252;
   1:  PR[GP1:91,2] = PR[GP1:90,2] + -0.493;
   1:L PR[91] R[100]mm/sec CNT100;
   1:  PR[GP1:91,1] = PR[GP1:90,1] + 0.513;
   1:  PR[GP1:91,2] = PR[GP1:90,2] + -0.504;
   1:L PR[91] R[100]mm/sec CNT100;
   1:  PR[GP1:91,1] = PR[GP1:90,1] + 3.796;
   1:  PR[GP1:91,2] = PR[GP1:90,2] + -1.803;
   1:L PR[91] R[100]mm/sec CNT100;
   1:  PR[GP1:91,1] = PR[GP1:90,1] + 3.992;
   1:  PR[GP1:91,2] = PR[GP1:90,2] + -2.159;
   1:L PR[91] R[100]mm/sec CNT100;
   1:  PR[GP1:91,1] = PR[GP1:90,1] + 4.061;
   1:  PR[GP1:91,2] = PR[GP1:90,2] + -2.221;
   1:L PR[91] R[100]mm/sec CNT100;
   1:  PR[GP1:91,1] = PR[GP1:90,1] + 4.295;
   1:  PR[GP1:91,2] = PR[GP1:90,2] + -2.603;
   1:L PR[91] R[100]mm/sec CNT100;
   1:  PR[GP1:91,1] = PR[GP1:90,1] + 5.671;
   1:  PR[GP1:91,2] = PR[GP1:90,2] + -5.144;
   1:L PR[91] R[100]mm/sec CNT100;
   1:  PR[GP1:91,1] = PR[GP1:90,1] + 5.719;
   1:  PR[GP1:91,2] = PR[GP1:90,2] + -5.583;
   1:L PR[91] R[100]mm/sec CNT100;
   1:  PR[GP1:91,1] = PR[GP1:90,1] + 5.858;
   1:  PR[GP1:91,2] = PR[GP1:90,2] + -6.143;
   1:L PR[91] R[100]mm/sec CNT100;
   1:  PR[GP1:91,1] = PR[GP1:90,1] + 8.932;
   1:  PR[GP1:91,2] = PR[GP1:90,2] + -15.414;
   1:L PR[91] R[100]mm/sec CNT100;
   1:  PR[GP1:91,1] = PR[GP1:90,1] + 9.372;
   1:  PR[GP1:91,2] = PR[GP1:90,2] + -16.371;
   1:L PR[91] R[100]mm/sec CNT100;
   1:  PR[GP1:91,1] = PR[GP1:90,1] + 9.995;
   1:  PR[GP1:91,2] = PR[GP1:90,2] + -17.248;
   1:L PR[91] R[100]mm/sec CNT100;
   1:  PR[GP1:91,1] = PR[GP1:90,1] + 15.664;
   1:  PR[GP1:91,2] = PR[GP1:90,2] + -24.672;
   1:L PR[91] R[100]mm/sec CNT100;
   1:  PR[GP1:91,1] = PR[GP1:90,1] + 16.654;
   1:  PR[GP1:91,2] = PR[GP1:90,2] + -25.624;
   1:L PR[91] R[100]mm/sec CNT100;
   1:  PR[GP1:91,1] = PR[GP1:90,1] + 25.177;
   1:  PR[GP1:91,2] = PR[GP1:90,2] + -31.266;
   1:L PR[91] R[100]mm/sec CNT100;
   1:  PR[GP1:91,1] = PR[GP1:90,1] + 26.796;
   1:  PR[GP1:91,2] = PR[GP1:90,2] + -31.935;
   1:L PR[91] R[100]mm/sec CNT100;
   1:  PR[GP1:91,1] = PR[GP1:90,1] + 28.582;
   1:  PR[GP1:91,2] = PR[GP1:90,2] + -32.307;
   1:L PR[91] R[100]mm/sec CNT100;
   1:  PR[GP1:91,1] = PR[GP1:90,1] + 36.518;
   1:  PR[GP1:91,2] = PR[GP1:90,2] + -34.363;
   1:L PR[91] R[100]mm/sec CNT100;
   1:  PR[GP1:91,1] = PR[GP1:90,1] + 38.671;
   1:  PR[GP1:91,2] = PR[GP1:90,2] + -34.402;
   1:L PR[91] R[100]mm/sec CNT100;
   1:  PR[GP1:91,1] = PR[GP1:90,1] + 45.906;
   1:  PR[GP1:91,2] = PR[GP1:90,2] + -33.858;
   1:L PR[91] R[100]mm/sec CNT100;
   1:  PR[GP1:91,1] = PR[GP1:90,1] + 48.375;
   1:  PR[GP1:91,2] = PR[GP1:90,2] + -33.437;
   1:L PR[91] R[100]mm/sec CNT100;
   1:  PR[GP1:91,1] = PR[GP1:90,1] + 50.734;
   1:  PR[GP1:91,2] = PR[GP1:90,2] + -32.561;
   1:L PR[91] R[100]mm/sec CNT100;
   1:  PR[GP1:91,1] = PR[GP1:90,1] + 56.958;
   1:  PR[GP1:91,2] = PR[GP1:90,2] + -29.880;
   1:L PR[91] R[100]mm/sec CNT100;
   1:  PR[GP1:91,1] = PR[GP1:90,1] + 59.318;
   1:  PR[GP1:91,2] = PR[GP1:90,2] + -28.457;
   1:L PR[91] R[100]mm/sec CNT100;
   1:  PR[GP1:91,1] = PR[GP1:90,1] + 61.402;
   1:  PR[GP1:91,2] = PR[GP1:90,2] + -26.594;
   1:L PR[91] R[100]mm/sec CNT100;
   1:  PR[GP1:91,1] = PR[GP1:90,1] + 66.126;
   1:  PR[GP1:91,2] = PR[GP1:90,2] + -22.287;
   1:L PR[91] R[100]mm/sec CNT100;
   1:  PR[GP1:91,1] = PR[GP1:90,1] + 67.911;
   1:  PR[GP1:91,2] = PR[GP1:90,2] + -19.961;
   1:L PR[91] R[100]mm/sec CNT100;
   1:  PR[GP1:91,1] = PR[GP1:90,1] + 69.260;
   1:  PR[GP1:91,2] = PR[GP1:90,2] + -17.287;
   1:L PR[91] R[100]mm/sec CNT100;
   1:  PR[GP1:91,1] = PR[GP1:90,1] + 72.185;
   1:  PR[GP1:91,2] = PR[GP1:90,2] + -11.923;
   1:L PR[91] R[100]mm/sec CNT100;
   1:  PR[GP1:91,1] = PR[GP1:90,1] + 73.023;
   1:  PR[GP1:91,2] = PR[GP1:90,2] + -9.010;
   1:L PR[91] R[100]mm/sec CNT100;
   1:  PR[GP1:91,1] = PR[GP1:90,1] + 73.315;
   1:  PR[GP1:91,2] = PR[GP1:90,2] + -5.905;
   1:L PR[91] R[100]mm/sec CNT100;
   1:  PR[GP1:91,1] = PR[GP1:90,1] + 74.291;
   1:  PR[GP1:91,2] = PR[GP1:90,2] + -0.050;
   1:L PR[91] R[100]mm/sec CNT100;
   1:  PR[GP1:91,1] = PR[GP1:90,1] + 73.995;
   1:  PR[GP1:91,2] = PR[GP1:90,2] + 3.110;
   1:L PR[91] R[100]mm/sec CNT100;
   1:  PR[GP1:91,1] = PR[GP1:90,1] + 73.030;
   1:  PR[GP1:91,2] = PR[GP1:90,2] + 8.845;
   1:L PR[91] R[100]mm/sec CNT100;
   1:  PR[GP1:91,1] = PR[GP1:90,1] + 72.182;
   1:  PR[GP1:91,2] = PR[GP1:90,2] + 11.788;
   1:L PR[91] R[100]mm/sec CNT100;
   1:  PR[GP1:91,1] = PR[GP1:90,1] + 70.791;
   1:  PR[GP1:91,2] = PR[GP1:90,2] + 14.544;
   1:L PR[91] R[100]mm/sec CNT100;
   1:  PR[GP1:91,1] = PR[GP1:90,1] + 67.917;
   1:  PR[GP1:91,2] = PR[GP1:90,2] + 19.809;
   1:L PR[91] R[100]mm/sec CNT100;
   1:  PR[GP1:91,1] = PR[GP1:90,1] + 66.128;
   1:  PR[GP1:91,2] = PR[GP1:90,2] + 22.141;
   1:L PR[91] R[100]mm/sec CNT100;
   1:  PR[GP1:91,1] = PR[GP1:90,1] + 63.900;
   1:  PR[GP1:91,2] = PR[GP1:90,2] + 24.133;
   1:L PR[91] R[100]mm/sec CNT100;
   1:  PR[GP1:91,1] = PR[GP1:90,1] + 59.316;
   1:  PR[GP1:91,2] = PR[GP1:90,2] + 28.315;
   1:L PR[91] R[100]mm/sec CNT100;
   1:  PR[GP1:91,1] = PR[GP1:90,1] + 56.971;
   1:  PR[GP1:91,2] = PR[GP1:90,2] + 29.728;
   1:L PR[91] R[100]mm/sec CNT100;
   1:  PR[GP1:91,1] = PR[GP1:90,1] + 54.334;
   1:  PR[GP1:91,2] = PR[GP1:90,2] + 30.708;
   1:L PR[91] R[100]mm/sec CNT100;
   1:  PR[GP1:91,1] = PR[GP1:90,1] + 48.359;
   1:  PR[GP1:91,2] = PR[GP1:90,2] + 33.296;
   1:L PR[91] R[100]mm/sec CNT100;
   1:  PR[GP1:91,1] = PR[GP1:90,1] + 45.906;
   1:  PR[GP1:91,2] = PR[GP1:90,2] + 33.714;
   1:L PR[91] R[100]mm/sec CNT100;
   1:  PR[GP1:91,1] = PR[GP1:90,1] + 38.671;
   1:  PR[GP1:91,2] = PR[GP1:90,2] + 34.258;
   1:L PR[91] R[100]mm/sec CNT100;
   1:  PR[GP1:91,1] = PR[GP1:90,1] + 36.503;
   1:  PR[GP1:91,2] = PR[GP1:90,2] + 34.219;
   1:L PR[91] R[100]mm/sec CNT100;
   1:  PR[GP1:91,1] = PR[GP1:90,1] + 34.368;
   1:  PR[GP1:91,2] = PR[GP1:90,2] + 33.774;
   1:L PR[91] R[100]mm/sec CNT100;
   1:  PR[GP1:91,1] = PR[GP1:90,1] + 26.810;
   1:  PR[GP1:91,2] = PR[GP1:90,2] + 31.797;
   1:L PR[91] R[100]mm/sec CNT100;
   1:  PR[GP1:91,1] = PR[GP1:90,1] + 25.175;
   1:  PR[GP1:91,2] = PR[GP1:90,2] + 31.121;
   1:L PR[91] R[100]mm/sec CNT100;
   1:  PR[GP1:91,1] = PR[GP1:90,1] + 23.663;
   1:  PR[GP1:91,2] = PR[GP1:90,2] + 30.133;
   1:L PR[91] R[100]mm/sec CNT100;
   1:  PR[GP1:91,1] = PR[GP1:90,1] + 16.654;
   1:  PR[GP1:91,2] = PR[GP1:90,2] + 25.480;
   1:L PR[91] R[100]mm/sec CNT100;
   1:  PR[GP1:91,1] = PR[GP1:90,1] + 15.671;
   1:  PR[GP1:91,2] = PR[GP1:90,2] + 24.535;
   1:L PR[91] R[100]mm/sec CNT100;
   1:  PR[GP1:91,1] = PR[GP1:90,1] + 14.844;
   1:  PR[GP1:91,2] = PR[GP1:90,2] + 23.371;
   1:L PR[91] R[100]mm/sec CNT100;
   1:  PR[GP1:91,1] = PR[GP1:90,1] + 9.367;
   1:  PR[GP1:91,2] = PR[GP1:90,2] + 16.217;
   1:L PR[91] R[100]mm/sec CNT100;
   1:  PR[GP1:91,1] = PR[GP1:90,1] + 8.932;
   1:  PR[GP1:91,2] = PR[GP1:90,2] + 15.270;
   1:L PR[91] R[100]mm/sec CNT100;
   1:  PR[GP1:91,1] = PR[GP1:90,1] + 5.858;
   1:  PR[GP1:91,2] = PR[GP1:90,2] + 5.997;
   1:L PR[91] R[100]mm/sec CNT100;
   1:  PR[GP1:91,1] = PR[GP1:90,1] + 5.721;
   1:  PR[GP1:91,2] = PR[GP1:90,2] + 5.445;
   1:L PR[91] R[100]mm/sec CNT100;
   1:  PR[GP1:91,1] = PR[GP1:90,1] + 5.675;
   1:  PR[GP1:91,2] = PR[GP1:90,2] + 5.030;
   1:L PR[91] R[100]mm/sec CNT100;
   1:  PR[GP1:91,1] = PR[GP1:90,1] + 4.901;
   1:  PR[GP1:91,2] = PR[GP1:90,2] + 3.186;
   1:L PR[91] R[100]mm/sec CNT100;
   1:  PR[GP1:91,1] = PR[GP1:90,1] + 4.536;
   1:  PR[GP1:91,2] = PR[GP1:90,2] + 2.507;
   1:L PR[91] R[100]mm/sec CNT100;
   1:  PR[GP1:91,1] = PR[GP1:90,1] + 3.820;
   1:  PR[GP1:91,2] = PR[GP1:90,2] + 1.730;
   1:L PR[91] R[100]mm/sec CNT100;
   1:  PR[GP1:91,1] = PR[GP1:90,1] + 2.725;
   1:  PR[GP1:91,2] = PR[GP1:90,2] + 0.975;
   1:L PR[91] R[100]mm/sec CNT100;
   1:  PR[GP1:91,1] = PR[GP1:90,1] + 2.309;
   1:  PR[GP1:91,2] = PR[GP1:90,2] + 0.838;
   1:L PR[91] R[100]mm/sec CNT100;
   1:  PR[GP1:91,1] = PR[GP1:90,1] + 0.051;
   1:  PR[GP1:91,2] = PR[GP1:90,2] + 0.300;
   1:L PR[91] R[100]mm/sec CNT100;
   1:  PR[GP1:91,1] = PR[GP1:90,1] + -0.073;
   1:  PR[GP1:91,2] = PR[GP1:90,2] + 0.350;
   1:L PR[91] R[100]mm/sec CNT100;
   1:  ! -- Layer/Ebene 24 -- !;
   1:  PR[91] = PR[90];
   1:  PR[GP1:91,1] = PR[GP1:90,1] + -3.401;
   1:  PR[GP1:91,2] = PR[GP1:90,2] + 1.622;
   1:  PR[GP1:91,3] = PR[GP1:90,3] + 14.945;
   1:L PR[91] R[100]mm/sec CNT100;
   1:  PR[GP1:91,1] = PR[GP1:90,1] + -3.653;
   1:  PR[GP1:91,2] = PR[GP1:90,2] + 1.828;
   1:L PR[91] R[100]mm/sec CNT100;
   1:  PR[GP1:91,1] = PR[GP1:90,1] + -4.080;
   1:  PR[GP1:91,2] = PR[GP1:90,2] + 2.580;
   1:L PR[91] R[100]mm/sec CNT100;
   1:  PR[GP1:91,1] = PR[GP1:90,1] + -5.391;
   1:  PR[GP1:91,2] = PR[GP1:90,2] + 5.000;
   1:L PR[91] R[100]mm/sec CNT100;
   1:  PR[GP1:91,1] = PR[GP1:90,1] + -5.422;
   1:  PR[GP1:91,2] = PR[GP1:90,2] + 5.290;
   1:L PR[91] R[100]mm/sec CNT100;
   1:  PR[GP1:91,1] = PR[GP1:90,1] + -5.463;
   1:  PR[GP1:91,2] = PR[GP1:90,2] + 5.455;
   1:L PR[91] R[100]mm/sec CNT100;
   1:  PR[GP1:91,1] = PR[GP1:90,1] + -8.850;
   1:  PR[GP1:91,2] = PR[GP1:90,2] + 15.676;
   1:L PR[91] R[100]mm/sec CNT100;
   1:  PR[GP1:91,1] = PR[GP1:90,1] + -9.062;
   1:  PR[GP1:91,2] = PR[GP1:90,2] + 16.137;
   1:L PR[91] R[100]mm/sec CNT100;
   1:  PR[GP1:91,1] = PR[GP1:90,1] + -9.370;
   1:  PR[GP1:91,2] = PR[GP1:90,2] + 16.570;
   1:L PR[91] R[100]mm/sec CNT100;
   1:  PR[GP1:91,1] = PR[GP1:90,1] + -15.616;
   1:  PR[GP1:91,2] = PR[GP1:90,2] + 24.747;
   1:L PR[91] R[100]mm/sec CNT100;
   1:  PR[GP1:91,1] = PR[GP1:90,1] + -16.237;
   1:  PR[GP1:91,2] = PR[GP1:90,2] + 25.344;
   1:L PR[91] R[100]mm/sec CNT100;
   1:  PR[GP1:91,1] = PR[GP1:90,1] + -25.079;
   1:  PR[GP1:91,2] = PR[GP1:90,2] + 31.201;
   1:L PR[91] R[100]mm/sec CNT100;
   1:  PR[GP1:91,1] = PR[GP1:90,1] + -26.261;
   1:  PR[GP1:91,2] = PR[GP1:90,2] + 31.690;
   1:L PR[91] R[100]mm/sec CNT100;
   1:  PR[GP1:91,1] = PR[GP1:90,1] + -27.586;
   1:  PR[GP1:91,2] = PR[GP1:90,2] + 31.966;
   1:L PR[91] R[100]mm/sec CNT100;
   1:  PR[GP1:91,1] = PR[GP1:90,1] + -36.329;
   1:  PR[GP1:91,2] = PR[GP1:90,2] + 34.230;
   1:L PR[91] R[100]mm/sec CNT100;
   1:  PR[GP1:91,1] = PR[GP1:90,1] + -38.050;
   1:  PR[GP1:91,2] = PR[GP1:90,2] + 34.261;
   1:L PR[91] R[100]mm/sec CNT100;
   1:  PR[GP1:91,1] = PR[GP1:90,1] + -46.022;
   1:  PR[GP1:91,2] = PR[GP1:90,2] + 33.661;
   1:L PR[91] R[100]mm/sec CNT100;
   1:  PR[GP1:91,1] = PR[GP1:90,1] + -48.097;
   1:  PR[GP1:91,2] = PR[GP1:90,2] + 33.308;
   1:L PR[91] R[100]mm/sec CNT100;
   1:  PR[GP1:91,1] = PR[GP1:90,1] + -50.082;
   1:  PR[GP1:91,2] = PR[GP1:90,2] + 32.570;
   1:L PR[91] R[100]mm/sec CNT100;
   1:  PR[GP1:91,1] = PR[GP1:90,1] + -56.940;
   1:  PR[GP1:91,2] = PR[GP1:90,2] + 29.616;
   1:L PR[91] R[100]mm/sec CNT100;
   1:  PR[GP1:91,1] = PR[GP1:90,1] + -58.982;
   1:  PR[GP1:91,2] = PR[GP1:90,2] + 28.384;
   1:L PR[91] R[100]mm/sec CNT100;
   1:  PR[GP1:91,1] = PR[GP1:90,1] + -60.788;
   1:  PR[GP1:91,2] = PR[GP1:90,2] + 26.770;
   1:L PR[91] R[100]mm/sec CNT100;
   1:  PR[GP1:91,1] = PR[GP1:90,1] + -65.995;
   1:  PR[GP1:91,2] = PR[GP1:90,2] + 22.025;
   1:L PR[91] R[100]mm/sec CNT100;
   1:  PR[GP1:91,1] = PR[GP1:90,1] + -67.564;
   1:  PR[GP1:91,2] = PR[GP1:90,2] + 19.979;
   1:L PR[91] R[100]mm/sec CNT100;
   1:  PR[GP1:91,1] = PR[GP1:90,1] + -68.754;
   1:  PR[GP1:91,2] = PR[GP1:90,2] + 17.621;
   1:L PR[91] R[100]mm/sec CNT100;
   1:  PR[GP1:91,1] = PR[GP1:90,1] + -71.977;
   1:  PR[GP1:91,2] = PR[GP1:90,2] + 11.705;
   1:L PR[91] R[100]mm/sec CNT100;
   1:  PR[GP1:91,1] = PR[GP1:90,1] + -72.721;
   1:  PR[GP1:91,2] = PR[GP1:90,2] + 9.121;
   1:L PR[91] R[100]mm/sec CNT100;
   1:  PR[GP1:91,1] = PR[GP1:90,1] + -72.980;
   1:  PR[GP1:91,2] = PR[GP1:90,2] + 6.356;
   1:L PR[91] R[100]mm/sec CNT100;
   1:  PR[GP1:91,1] = PR[GP1:90,1] + -74.056;
   1:  PR[GP1:91,2] = PR[GP1:90,2] + -0.094;
   1:L PR[91] R[100]mm/sec CNT100;
   1:  PR[GP1:91,1] = PR[GP1:90,1] + -73.791;
   1:  PR[GP1:91,2] = PR[GP1:90,2] + -2.926;
   1:L PR[91] R[100]mm/sec CNT100;
   1:  PR[GP1:91,1] = PR[GP1:90,1] + -72.727;
   1:  PR[GP1:91,2] = PR[GP1:90,2] + -9.243;
   1:L PR[91] R[100]mm/sec CNT100;
   1:  PR[GP1:91,1] = PR[GP1:90,1] + -71.974;
   1:  PR[GP1:91,2] = PR[GP1:90,2] + -11.858;
   1:L PR[91] R[100]mm/sec CNT100;
   1:  PR[GP1:91,1] = PR[GP1:90,1] + -70.737;
   1:  PR[GP1:91,2] = PR[GP1:90,2] + -14.309;
   1:L PR[91] R[100]mm/sec CNT100;
   1:  PR[GP1:91,1] = PR[GP1:90,1] + -67.570;
   1:  PR[GP1:91,2] = PR[GP1:90,2] + -20.115;
   1:L PR[91] R[100]mm/sec CNT100;
   1:  PR[GP1:91,1] = PR[GP1:90,1] + -65.996;
   1:  PR[GP1:91,2] = PR[GP1:90,2] + -22.167;
   1:L PR[91] R[100]mm/sec CNT100;
   1:  PR[GP1:91,1] = PR[GP1:90,1] + -64.032;
   1:  PR[GP1:91,2] = PR[GP1:90,2] + -23.924;
   1:L PR[91] R[100]mm/sec CNT100;
   1:  PR[GP1:91,1] = PR[GP1:90,1] + -58.980;
   1:  PR[GP1:91,2] = PR[GP1:90,2] + -28.530;
   1:L PR[91] R[100]mm/sec CNT100;
   1:  PR[GP1:91,1] = PR[GP1:90,1] + -56.954;
   1:  PR[GP1:91,2] = PR[GP1:90,2] + -29.752;
   1:L PR[91] R[100]mm/sec CNT100;
   1:  PR[GP1:91,1] = PR[GP1:90,1] + -54.666;
   1:  PR[GP1:91,2] = PR[GP1:90,2] + -30.602;
   1:L PR[91] R[100]mm/sec CNT100;
   1:  PR[GP1:91,1] = PR[GP1:90,1] + -48.081;
   1:  PR[GP1:91,2] = PR[GP1:90,2] + -33.454;
   1:L PR[91] R[100]mm/sec CNT100;
   1:  PR[GP1:91,1] = PR[GP1:90,1] + -46.022;
   1:  PR[GP1:91,2] = PR[GP1:90,2] + -33.805;
   1:L PR[91] R[100]mm/sec CNT100;
   1:  PR[GP1:91,1] = PR[GP1:90,1] + -38.050;
   1:  PR[GP1:91,2] = PR[GP1:90,2] + -34.405;
   1:L PR[91] R[100]mm/sec CNT100;
   1:  PR[GP1:91,1] = PR[GP1:90,1] + -36.315;
   1:  PR[GP1:91,2] = PR[GP1:90,2] + -34.374;
   1:L PR[91] R[100]mm/sec CNT100;
   1:  PR[GP1:91,1] = PR[GP1:90,1] + -34.603;
   1:  PR[GP1:91,2] = PR[GP1:90,2] + -34.018;
   1:L PR[91] R[100]mm/sec CNT100;
   1:  PR[GP1:91,1] = PR[GP1:90,1] + -26.276;
   1:  PR[GP1:91,2] = PR[GP1:90,2] + -31.840;
   1:L PR[91] R[100]mm/sec CNT100;
   1:  PR[GP1:91,1] = PR[GP1:90,1] + -25.079;
   1:  PR[GP1:91,2] = PR[GP1:90,2] + -31.345;
   1:L PR[91] R[100]mm/sec CNT100;
   1:  PR[GP1:91,1] = PR[GP1:90,1] + -16.237;
   1:  PR[GP1:91,2] = PR[GP1:90,2] + -25.488;
   1:L PR[91] R[100]mm/sec CNT100;
   1:  PR[GP1:91,1] = PR[GP1:90,1] + -15.624;
   1:  PR[GP1:91,2] = PR[GP1:90,2] + -24.898;
   1:L PR[91] R[100]mm/sec CNT100;
   1:  PR[GP1:91,1] = PR[GP1:90,1] + -15.093;
   1:  PR[GP1:91,2] = PR[GP1:90,2] + -24.151;
   1:L PR[91] R[100]mm/sec CNT100;
   1:  PR[GP1:91,1] = PR[GP1:90,1] + -9.058;
   1:  PR[GP1:91,2] = PR[GP1:90,2] + -16.271;
   1:L PR[91] R[100]mm/sec CNT100;
   1:  PR[GP1:91,1] = PR[GP1:90,1] + -8.850;
   1:  PR[GP1:91,2] = PR[GP1:90,2] + -15.820;
   1:L PR[91] R[100]mm/sec CNT100;
   1:  PR[GP1:91,1] = PR[GP1:90,1] + -5.464;
   1:  PR[GP1:91,2] = PR[GP1:90,2] + -5.601;
   1:L PR[91] R[100]mm/sec CNT100;
   1:  PR[GP1:91,1] = PR[GP1:90,1] + -5.423;
   1:  PR[GP1:91,2] = PR[GP1:90,2] + -5.438;
   1:L PR[91] R[100]mm/sec CNT100;
   1:  PR[GP1:91,1] = PR[GP1:90,1] + -5.394;
   1:  PR[GP1:91,2] = PR[GP1:90,2] + -5.173;
   1:L PR[91] R[100]mm/sec CNT100;
   1:  PR[GP1:91,1] = PR[GP1:90,1] + -4.364;
   1:  PR[GP1:91,2] = PR[GP1:90,2] + -2.744;
   1:L PR[91] R[100]mm/sec CNT100;
   1:  PR[GP1:91,1] = PR[GP1:90,1] + -3.550;
   1:  PR[GP1:91,2] = PR[GP1:90,2] + -1.860;
   1:L PR[91] R[100]mm/sec CNT100;
   1:  PR[GP1:91,1] = PR[GP1:90,1] + -2.129;
   1:  PR[GP1:91,2] = PR[GP1:90,2] + -1.044;
   1:L PR[91] R[100]mm/sec CNT100;
   1:  PR[GP1:91,1] = PR[GP1:90,1] + -0.081;
   1:  PR[GP1:91,2] = PR[GP1:90,2] + -0.590;
   1:L PR[91] R[100]mm/sec CNT100;
   1:  PR[GP1:91,1] = PR[GP1:90,1] + 0.253;
   1:  PR[GP1:91,2] = PR[GP1:90,2] + -0.588;
   1:L PR[91] R[100]mm/sec CNT100;
   1:  PR[GP1:91,1] = PR[GP1:90,1] + 3.614;
   1:  PR[GP1:91,2] = PR[GP1:90,2] + -1.766;
   1:L PR[91] R[100]mm/sec CNT100;
   1:  PR[GP1:91,1] = PR[GP1:90,1] + 3.866;
   1:  PR[GP1:91,2] = PR[GP1:90,2] + -1.973;
   1:L PR[91] R[100]mm/sec CNT100;
   1:  PR[GP1:91,1] = PR[GP1:90,1] + 4.289;
   1:  PR[GP1:91,2] = PR[GP1:90,2] + -2.717;
   1:L PR[91] R[100]mm/sec CNT100;
   1:  PR[GP1:91,1] = PR[GP1:90,1] + 5.604;
   1:  PR[GP1:91,2] = PR[GP1:90,2] + -5.145;
   1:L PR[91] R[100]mm/sec CNT100;
   1:  PR[GP1:91,1] = PR[GP1:90,1] + 5.635;
   1:  PR[GP1:91,2] = PR[GP1:90,2] + -5.436;
   1:L PR[91] R[100]mm/sec CNT100;
   1:  PR[GP1:91,1] = PR[GP1:90,1] + 5.676;
   1:  PR[GP1:91,2] = PR[GP1:90,2] + -5.602;
   1:L PR[91] R[100]mm/sec CNT100;
   1:  PR[GP1:91,1] = PR[GP1:90,1] + 9.062;
   1:  PR[GP1:91,2] = PR[GP1:90,2] + -15.816;
   1:L PR[91] R[100]mm/sec CNT100;
   1:  PR[GP1:91,1] = PR[GP1:90,1] + 9.274;
   1:  PR[GP1:91,2] = PR[GP1:90,2] + -16.277;
   1:L PR[91] R[100]mm/sec CNT100;
   1:  PR[GP1:91,1] = PR[GP1:90,1] + 9.582;
   1:  PR[GP1:91,2] = PR[GP1:90,2] + -16.710;
   1:L PR[91] R[100]mm/sec CNT100;
   1:  PR[GP1:91,1] = PR[GP1:90,1] + 15.828;
   1:  PR[GP1:91,2] = PR[GP1:90,2] + -24.890;
   1:L PR[91] R[100]mm/sec CNT100;
   1:  PR[GP1:91,1] = PR[GP1:90,1] + 16.448;
   1:  PR[GP1:91,2] = PR[GP1:90,2] + -25.487;
   1:L PR[91] R[100]mm/sec CNT100;
   1:  PR[GP1:91,1] = PR[GP1:90,1] + 25.290;
   1:  PR[GP1:91,2] = PR[GP1:90,2] + -31.344;
   1:L PR[91] R[100]mm/sec CNT100;
   1:  PR[GP1:91,1] = PR[GP1:90,1] + 26.473;
   1:  PR[GP1:91,2] = PR[GP1:90,2] + -31.833;
   1:L PR[91] R[100]mm/sec CNT100;
   1:  PR[GP1:91,1] = PR[GP1:90,1] + 27.797;
   1:  PR[GP1:91,2] = PR[GP1:90,2] + -32.109;
   1:L PR[91] R[100]mm/sec CNT100;
   1:  PR[GP1:91,1] = PR[GP1:90,1] + 36.541;
   1:  PR[GP1:91,2] = PR[GP1:90,2] + -34.374;
   1:L PR[91] R[100]mm/sec CNT100;
   1:  PR[GP1:91,1] = PR[GP1:90,1] + 38.261;
   1:  PR[GP1:91,2] = PR[GP1:90,2] + -34.405;
   1:L PR[91] R[100]mm/sec CNT100;
   1:  PR[GP1:91,1] = PR[GP1:90,1] + 46.234;
   1:  PR[GP1:91,2] = PR[GP1:90,2] + -33.805;
   1:L PR[91] R[100]mm/sec CNT100;
   1:  PR[GP1:91,1] = PR[GP1:90,1] + 48.309;
   1:  PR[GP1:91,2] = PR[GP1:90,2] + -33.452;
   1:L PR[91] R[100]mm/sec CNT100;
   1:  PR[GP1:91,1] = PR[GP1:90,1] + 50.294;
   1:  PR[GP1:91,2] = PR[GP1:90,2] + -32.714;
   1:L PR[91] R[100]mm/sec CNT100;
   1:  PR[GP1:91,1] = PR[GP1:90,1] + 57.153;
   1:  PR[GP1:91,2] = PR[GP1:90,2] + -29.761;
   1:L PR[91] R[100]mm/sec CNT100;
   1:  PR[GP1:91,1] = PR[GP1:90,1] + 59.195;
   1:  PR[GP1:91,2] = PR[GP1:90,2] + -28.529;
   1:L PR[91] R[100]mm/sec CNT100;
   1:  PR[GP1:91,1] = PR[GP1:90,1] + 61.000;
   1:  PR[GP1:91,2] = PR[GP1:90,2] + -26.915;
   1:L PR[91] R[100]mm/sec CNT100;
   1:  PR[GP1:91,1] = PR[GP1:90,1] + 66.207;
   1:  PR[GP1:91,2] = PR[GP1:90,2] + -22.168;
   1:L PR[91] R[100]mm/sec CNT100;
   1:  PR[GP1:91,1] = PR[GP1:90,1] + 67.777;
   1:  PR[GP1:91,2] = PR[GP1:90,2] + -20.122;
   1:L PR[91] R[100]mm/sec CNT100;
   1:  PR[GP1:91,1] = PR[GP1:90,1] + 68.967;
   1:  PR[GP1:91,2] = PR[GP1:90,2] + -17.764;
   1:L PR[91] R[100]mm/sec CNT100;
   1:  PR[GP1:91,1] = PR[GP1:90,1] + 72.190;
   1:  PR[GP1:91,2] = PR[GP1:90,2] + -11.852;
   1:L PR[91] R[100]mm/sec CNT100;
   1:  PR[GP1:91,1] = PR[GP1:90,1] + 72.934;
   1:  PR[GP1:91,2] = PR[GP1:90,2] + -9.267;
   1:L PR[91] R[100]mm/sec CNT100;
   1:  PR[GP1:91,1] = PR[GP1:90,1] + 73.193;
   1:  PR[GP1:91,2] = PR[GP1:90,2] + -6.503;
   1:L PR[91] R[100]mm/sec CNT100;
   1:  PR[GP1:91,1] = PR[GP1:90,1] + 74.269;
   1:  PR[GP1:91,2] = PR[GP1:90,2] + -0.050;
   1:L PR[91] R[100]mm/sec CNT100;
   1:  PR[GP1:91,1] = PR[GP1:90,1] + 74.004;
   1:  PR[GP1:91,2] = PR[GP1:90,2] + 2.782;
   1:L PR[91] R[100]mm/sec CNT100;
   1:  PR[GP1:91,1] = PR[GP1:90,1] + 72.940;
   1:  PR[GP1:91,2] = PR[GP1:90,2] + 9.102;
   1:L PR[91] R[100]mm/sec CNT100;
   1:  PR[GP1:91,1] = PR[GP1:90,1] + 72.187;
   1:  PR[GP1:91,2] = PR[GP1:90,2] + 11.717;
   1:L PR[91] R[100]mm/sec CNT100;
   1:  PR[GP1:91,1] = PR[GP1:90,1] + 70.951;
   1:  PR[GP1:91,2] = PR[GP1:90,2] + 14.168;
   1:L PR[91] R[100]mm/sec CNT100;
   1:  PR[GP1:91,1] = PR[GP1:90,1] + 67.783;
   1:  PR[GP1:91,2] = PR[GP1:90,2] + 19.970;
   1:L PR[91] R[100]mm/sec CNT100;
   1:  PR[GP1:91,1] = PR[GP1:90,1] + 66.209;
   1:  PR[GP1:91,2] = PR[GP1:90,2] + 22.022;
   1:L PR[91] R[100]mm/sec CNT100;
   1:  PR[GP1:91,1] = PR[GP1:90,1] + 64.245;
   1:  PR[GP1:91,2] = PR[GP1:90,2] + 23.779;
   1:L PR[91] R[100]mm/sec CNT100;
   1:  PR[GP1:91,1] = PR[GP1:90,1] + 59.192;
   1:  PR[GP1:91,2] = PR[GP1:90,2] + 28.387;
   1:L PR[91] R[100]mm/sec CNT100;
   1:  PR[GP1:91,1] = PR[GP1:90,1] + 57.166;
   1:  PR[GP1:91,2] = PR[GP1:90,2] + 29.609;
   1:L PR[91] R[100]mm/sec CNT100;
   1:  PR[GP1:91,1] = PR[GP1:90,1] + 54.878;
   1:  PR[GP1:91,2] = PR[GP1:90,2] + 30.459;
   1:L PR[91] R[100]mm/sec CNT100;
   1:  PR[GP1:91,1] = PR[GP1:90,1] + 48.293;
   1:  PR[GP1:91,2] = PR[GP1:90,2] + 33.310;
   1:L PR[91] R[100]mm/sec CNT100;
   1:  PR[GP1:91,1] = PR[GP1:90,1] + 46.234;
   1:  PR[GP1:91,2] = PR[GP1:90,2] + 33.661;
   1:L PR[91] R[100]mm/sec CNT100;
   1:  PR[GP1:91,1] = PR[GP1:90,1] + 38.261;
   1:  PR[GP1:91,2] = PR[GP1:90,2] + 34.261;
   1:L PR[91] R[100]mm/sec CNT100;
   1:  PR[GP1:91,1] = PR[GP1:90,1] + 36.526;
   1:  PR[GP1:91,2] = PR[GP1:90,2] + 34.230;
   1:L PR[91] R[100]mm/sec CNT100;
   1:  PR[GP1:91,1] = PR[GP1:90,1] + 34.815;
   1:  PR[GP1:91,2] = PR[GP1:90,2] + 33.874;
   1:L PR[91] R[100]mm/sec CNT100;
   1:  PR[GP1:91,1] = PR[GP1:90,1] + 26.487;
   1:  PR[GP1:91,2] = PR[GP1:90,2] + 31.695;
   1:L PR[91] R[100]mm/sec CNT100;
   1:  PR[GP1:91,1] = PR[GP1:90,1] + 25.290;
   1:  PR[GP1:91,2] = PR[GP1:90,2] + 31.200;
   1:L PR[91] R[100]mm/sec CNT100;
   1:  PR[GP1:91,1] = PR[GP1:90,1] + 16.448;
   1:  PR[GP1:91,2] = PR[GP1:90,2] + 25.343;
   1:L PR[91] R[100]mm/sec CNT100;
   1:  PR[GP1:91,1] = PR[GP1:90,1] + 15.835;
   1:  PR[GP1:91,2] = PR[GP1:90,2] + 24.753;
   1:L PR[91] R[100]mm/sec CNT100;
   1:  PR[GP1:91,1] = PR[GP1:90,1] + 15.305;
   1:  PR[GP1:91,2] = PR[GP1:90,2] + 24.006;
   1:L PR[91] R[100]mm/sec CNT100;
   1:  PR[GP1:91,1] = PR[GP1:90,1] + 9.270;
   1:  PR[GP1:91,2] = PR[GP1:90,2] + 16.123;
   1:L PR[91] R[100]mm/sec CNT100;
   1:  PR[GP1:91,1] = PR[GP1:90,1] + 9.062;
   1:  PR[GP1:91,2] = PR[GP1:90,2] + 15.672;
   1:L PR[91] R[100]mm/sec CNT100;
   1:  PR[GP1:91,1] = PR[GP1:90,1] + 5.676;
   1:  PR[GP1:91,2] = PR[GP1:90,2] + 5.455;
   1:L PR[91] R[100]mm/sec CNT100;
   1:  PR[GP1:91,1] = PR[GP1:90,1] + 5.636;
   1:  PR[GP1:91,2] = PR[GP1:90,2] + 5.293;
   1:L PR[91] R[100]mm/sec CNT100;
   1:  PR[GP1:91,1] = PR[GP1:90,1] + 5.607;
   1:  PR[GP1:91,2] = PR[GP1:90,2] + 5.030;
   1:L PR[91] R[100]mm/sec CNT100;
   1:  PR[GP1:91,1] = PR[GP1:90,1] + 4.578;
   1:  PR[GP1:91,2] = PR[GP1:90,2] + 2.601;
   1:L PR[91] R[100]mm/sec CNT100;
   1:  PR[GP1:91,1] = PR[GP1:90,1] + 3.763;
   1:  PR[GP1:91,2] = PR[GP1:90,2] + 1.716;
   1:L PR[91] R[100]mm/sec CNT100;
   1:  PR[GP1:91,1] = PR[GP1:90,1] + 2.342;
   1:  PR[GP1:91,2] = PR[GP1:90,2] + 0.901;
   1:L PR[91] R[100]mm/sec CNT100;
   1:  PR[GP1:91,1] = PR[GP1:90,1] + 0.295;
   1:  PR[GP1:91,2] = PR[GP1:90,2] + 0.446;
   1:L PR[91] R[100]mm/sec CNT100;
   1:  PR[GP1:91,1] = PR[GP1:90,1] + -0.040;
   1:  PR[GP1:91,2] = PR[GP1:90,2] + 0.444;
   1:L PR[91] R[100]mm/sec CNT100;
   1:  ! -- Layer/Ebene 25 -- !;
   1:  PR[91] = PR[90];
   1:  PR[GP1:91,1] = PR[GP1:90,1] + -3.219;
   1:  PR[GP1:91,2] = PR[GP1:90,2] + 1.776;
   1:  PR[GP1:91,3] = PR[GP1:90,3] + 15.555;
   1:L PR[91] R[100]mm/sec CNT100;
   1:  PR[GP1:91,1] = PR[GP1:90,1] + -3.450;
   1:  PR[GP1:91,2] = PR[GP1:90,2] + 1.964;
   1:L PR[91] R[100]mm/sec CNT100;
   1:  PR[GP1:91,1] = PR[GP1:90,1] + -5.322;
   1:  PR[GP1:91,2] = PR[GP1:90,2] + 5.253;
   1:L PR[91] R[100]mm/sec CNT100;
   1:  PR[GP1:91,1] = PR[GP1:90,1] + -8.980;
   1:  PR[GP1:91,2] = PR[GP1:90,2] + 16.060;
   1:L PR[91] R[100]mm/sec CNT100;
   1:  PR[GP1:91,1] = PR[GP1:90,1] + -15.780;
   1:  PR[GP1:91,2] = PR[GP1:90,2] + 24.964;
   1:L PR[91] R[100]mm/sec CNT100;
   1:  PR[GP1:91,1] = PR[GP1:90,1] + -16.032;
   1:  PR[GP1:91,2] = PR[GP1:90,2] + 25.207;
   1:L PR[91] R[100]mm/sec CNT100;
   1:  PR[GP1:91,1] = PR[GP1:90,1] + -25.192;
   1:  PR[GP1:91,2] = PR[GP1:90,2] + 31.279;
   1:L PR[91] R[100]mm/sec CNT100;
   1:  PR[GP1:91,1] = PR[GP1:90,1] + -25.939;
   1:  PR[GP1:91,2] = PR[GP1:90,2] + 31.588;
   1:L PR[91] R[100]mm/sec CNT100;
   1:  PR[GP1:91,1] = PR[GP1:90,1] + -26.801;
   1:  PR[GP1:91,2] = PR[GP1:90,2] + 31.767;
   1:L PR[91] R[100]mm/sec CNT100;
   1:  PR[GP1:91,1] = PR[GP1:90,1] + -36.353;
   1:  PR[GP1:91,2] = PR[GP1:90,2] + 34.241;
   1:L PR[91] R[100]mm/sec CNT100;
   1:  PR[GP1:91,1] = PR[GP1:90,1] + -37.640;
   1:  PR[GP1:91,2] = PR[GP1:90,2] + 34.264;
   1:L PR[91] R[100]mm/sec CNT100;
   1:  PR[GP1:91,1] = PR[GP1:90,1] + -46.350;
   1:  PR[GP1:91,2] = PR[GP1:90,2] + 33.609;
   1:L PR[91] R[100]mm/sec CNT100;
   1:  PR[GP1:91,1] = PR[GP1:90,1] + -48.032;
   1:  PR[GP1:91,2] = PR[GP1:90,2] + 33.322;
   1:L PR[91] R[100]mm/sec CNT100;
   1:  PR[GP1:91,1] = PR[GP1:90,1] + -49.643;
   1:  PR[GP1:91,2] = PR[GP1:90,2] + 32.724;
   1:L PR[91] R[100]mm/sec CNT100;
   1:  PR[GP1:91,1] = PR[GP1:90,1] + -57.136;
   1:  PR[GP1:91,2] = PR[GP1:90,2] + 29.496;
   1:L PR[91] R[100]mm/sec CNT100;
   1:  PR[GP1:91,1] = PR[GP1:90,1] + -58.859;
   1:  PR[GP1:91,2] = PR[GP1:90,2] + 28.457;
   1:L PR[91] R[100]mm/sec CNT100;
   1:  PR[GP1:91,1] = PR[GP1:90,1] + -60.387;
   1:  PR[GP1:91,2] = PR[GP1:90,2] + 27.090;
   1:L PR[91] R[100]mm/sec CNT100;
   1:  PR[GP1:91,1] = PR[GP1:90,1] + -66.076;
   1:  PR[GP1:91,2] = PR[GP1:90,2] + 21.906;
   1:L PR[91] R[100]mm/sec CNT100;
   1:  PR[GP1:91,1] = PR[GP1:90,1] + -67.430;
   1:  PR[GP1:91,2] = PR[GP1:90,2] + 20.140;
   1:L PR[91] R[100]mm/sec CNT100;
   1:  PR[GP1:91,1] = PR[GP1:90,1] + -68.461;
   1:  PR[GP1:91,2] = PR[GP1:90,2] + 18.097;
   1:L PR[91] R[100]mm/sec CNT100;
   1:  PR[GP1:91,1] = PR[GP1:90,1] + -71.982;
   1:  PR[GP1:91,2] = PR[GP1:90,2] + 11.634;
   1:L PR[91] R[100]mm/sec CNT100;
   1:  PR[GP1:91,1] = PR[GP1:90,1] + -72.632;
   1:  PR[GP1:91,2] = PR[GP1:90,2] + 9.378;
   1:L PR[91] R[100]mm/sec CNT100;
   1:  PR[GP1:91,1] = PR[GP1:90,1] + -72.859;
   1:  PR[GP1:91,2] = PR[GP1:90,2] + 6.954;
   1:L PR[91] R[100]mm/sec CNT100;
   1:  PR[GP1:91,1] = PR[GP1:90,1] + -74.035;
   1:  PR[GP1:91,2] = PR[GP1:90,2] + -0.094;
   1:L PR[91] R[100]mm/sec CNT100;
   1:  PR[GP1:91,1] = PR[GP1:90,1] + -73.800;
   1:  PR[GP1:91,2] = PR[GP1:90,2] + -2.598;
   1:L PR[91] R[100]mm/sec CNT100;
   1:  PR[GP1:91,1] = PR[GP1:90,1] + -72.638;
   1:  PR[GP1:91,2] = PR[GP1:90,2] + -9.501;
   1:L PR[91] R[100]mm/sec CNT100;
   1:  PR[GP1:91,1] = PR[GP1:90,1] + -71.980;
   1:  PR[GP1:91,2] = PR[GP1:90,2] + -11.787;
   1:L PR[91] R[100]mm/sec CNT100;
   1:  PR[GP1:91,1] = PR[GP1:90,1] + -70.897;
   1:  PR[GP1:91,2] = PR[GP1:90,2] + -13.933;
   1:L PR[91] R[100]mm/sec CNT100;
   1:  PR[GP1:91,1] = PR[GP1:90,1] + -67.436;
   1:  PR[GP1:91,2] = PR[GP1:90,2] + -20.277;
   1:L PR[91] R[100]mm/sec CNT100;
   1:  PR[GP1:91,1] = PR[GP1:90,1] + -66.077;
   1:  PR[GP1:91,2] = PR[GP1:90,2] + -22.048;
   1:L PR[91] R[100]mm/sec CNT100;
   1:  PR[GP1:91,1] = PR[GP1:90,1] + -64.376;
   1:  PR[GP1:91,2] = PR[GP1:90,2] + -23.569;
   1:L PR[91] R[100]mm/sec CNT100;
   1:  PR[GP1:91,1] = PR[GP1:90,1] + -58.856;
   1:  PR[GP1:91,2] = PR[GP1:90,2] + -28.602;
   1:L PR[91] R[100]mm/sec CNT100;
   1:  PR[GP1:91,1] = PR[GP1:90,1] + -57.149;
   1:  PR[GP1:91,2] = PR[GP1:90,2] + -29.632;
   1:L PR[91] R[100]mm/sec CNT100;
   1:  PR[GP1:91,1] = PR[GP1:90,1] + -55.210;
   1:  PR[GP1:91,2] = PR[GP1:90,2] + -30.352;
   1:L PR[91] R[100]mm/sec CNT100;
   1:  PR[GP1:91,1] = PR[GP1:90,1] + -48.016;
   1:  PR[GP1:91,2] = PR[GP1:90,2] + -33.469;
   1:L PR[91] R[100]mm/sec CNT100;
   1:  PR[GP1:91,1] = PR[GP1:90,1] + -46.350;
   1:  PR[GP1:91,2] = PR[GP1:90,2] + -33.753;
   1:L PR[91] R[100]mm/sec CNT100;
   1:  PR[GP1:91,1] = PR[GP1:90,1] + -37.640;
   1:  PR[GP1:91,2] = PR[GP1:90,2] + -34.408;
   1:L PR[91] R[100]mm/sec CNT100;
   1:  PR[GP1:91,1] = PR[GP1:90,1] + -36.338;
   1:  PR[GP1:91,2] = PR[GP1:90,2] + -34.384;
   1:L PR[91] R[100]mm/sec CNT100;
   1:  PR[GP1:91,1] = PR[GP1:90,1] + -35.051;
   1:  PR[GP1:91,2] = PR[GP1:90,2] + -34.117;
   1:L PR[91] R[100]mm/sec CNT100;
   1:  PR[GP1:91,1] = PR[GP1:90,1] + -25.953;
   1:  PR[GP1:91,2] = PR[GP1:90,2] + -31.738;
   1:L PR[91] R[100]mm/sec CNT100;
   1:  PR[GP1:91,1] = PR[GP1:90,1] + -25.192;
   1:  PR[GP1:91,2] = PR[GP1:90,2] + -31.423;
   1:L PR[91] R[100]mm/sec CNT100;
   1:  PR[GP1:91,1] = PR[GP1:90,1] + -16.032;
   1:  PR[GP1:91,2] = PR[GP1:90,2] + -25.351;
   1:L PR[91] R[100]mm/sec CNT100;
   1:  PR[GP1:91,1] = PR[GP1:90,1] + -15.788;
   1:  PR[GP1:91,2] = PR[GP1:90,2] + -25.115;
   1:L PR[91] R[100]mm/sec CNT100;
   1:  PR[GP1:91,1] = PR[GP1:90,1] + -15.553;
   1:  PR[GP1:91,2] = PR[GP1:90,2] + -24.786;
   1:L PR[91] R[100]mm/sec CNT100;
   1:  PR[GP1:91,1] = PR[GP1:90,1] + -8.980;
   1:  PR[GP1:91,2] = PR[GP1:90,2] + -16.204;
   1:L PR[91] R[100]mm/sec CNT100;
   1:  PR[GP1:91,1] = PR[GP1:90,1] + -5.339;
   1:  PR[GP1:91,2] = PR[GP1:90,2] + -5.446;
   1:L PR[91] R[100]mm/sec CNT100;
   1:  PR[GP1:91,1] = PR[GP1:90,1] + -5.056;
   1:  PR[GP1:91,2] = PR[GP1:90,2] + -4.653;
   1:L PR[91] R[100]mm/sec CNT100;
   1:  PR[GP1:91,1] = PR[GP1:90,1] + -4.349;
   1:  PR[GP1:91,2] = PR[GP1:90,2] + -2.990;
   1:L PR[91] R[100]mm/sec CNT100;
   1:  PR[GP1:91,1] = PR[GP1:90,1] + -3.895;
   1:  PR[GP1:91,2] = PR[GP1:90,2] + -2.590;
   1:L PR[91] R[100]mm/sec CNT100;
   1:  PR[GP1:91,1] = PR[GP1:90,1] + -3.276;
   1:  PR[GP1:91,2] = PR[GP1:90,2] + -1.953;
   1:L PR[91] R[100]mm/sec CNT100;
   1:  PR[GP1:91,1] = PR[GP1:90,1] + -2.327;
   1:  PR[GP1:91,2] = PR[GP1:90,2] + -1.481;
   1:L PR[91] R[100]mm/sec CNT100;
   1:  PR[GP1:91,1] = PR[GP1:90,1] + -1.497;
   1:  PR[GP1:91,2] = PR[GP1:90,2] + -1.010;
   1:L PR[91] R[100]mm/sec CNT100;
   1:  PR[GP1:91,1] = PR[GP1:90,1] + -0.221;
   1:  PR[GP1:91,2] = PR[GP1:90,2] + -0.726;
   1:L PR[91] R[100]mm/sec CNT100;
   1:  PR[GP1:91,1] = PR[GP1:90,1] + 0.047;
   1:  PR[GP1:91,2] = PR[GP1:90,2] + -0.725;
   1:L PR[91] R[100]mm/sec CNT100;
   1:  PR[GP1:91,1] = PR[GP1:90,1] + 3.433;
   1:  PR[GP1:91,2] = PR[GP1:90,2] + -1.920;
   1:L PR[91] R[100]mm/sec CNT100;
   1:  PR[GP1:91,1] = PR[GP1:90,1] + 3.663;
   1:  PR[GP1:91,2] = PR[GP1:90,2] + -2.109;
   1:L PR[91] R[100]mm/sec CNT100;
   1:  PR[GP1:91,1] = PR[GP1:90,1] + 5.068;
   1:  PR[GP1:91,2] = PR[GP1:90,2] + -4.582;
   1:L PR[91] R[100]mm/sec CNT100;
   1:  PR[GP1:91,1] = PR[GP1:90,1] + 5.390;
   1:  PR[GP1:91,2] = PR[GP1:90,2] + -5.194;
   1:L PR[91] R[100]mm/sec CNT100;
   1:  PR[GP1:91,1] = PR[GP1:90,1] + 5.516;
   1:  PR[GP1:91,2] = PR[GP1:90,2] + -5.343;
   1:L PR[91] R[100]mm/sec CNT100;
   1:  PR[GP1:91,1] = PR[GP1:90,1] + 9.192;
   1:  PR[GP1:91,2] = PR[GP1:90,2] + -16.200;
   1:L PR[91] R[100]mm/sec CNT100;
   1:  PR[GP1:91,1] = PR[GP1:90,1] + 15.992;
   1:  PR[GP1:91,2] = PR[GP1:90,2] + -25.107;
   1:L PR[91] R[100]mm/sec CNT100;
   1:  PR[GP1:91,1] = PR[GP1:90,1] + 16.243;
   1:  PR[GP1:91,2] = PR[GP1:90,2] + -25.349;
   1:L PR[91] R[100]mm/sec CNT100;
   1:  PR[GP1:91,1] = PR[GP1:90,1] + 25.404;
   1:  PR[GP1:91,2] = PR[GP1:90,2] + -31.422;
   1:L PR[91] R[100]mm/sec CNT100;
   1:  PR[GP1:91,1] = PR[GP1:90,1] + 26.150;
   1:  PR[GP1:91,2] = PR[GP1:90,2] + -31.731;
   1:L PR[91] R[100]mm/sec CNT100;
   1:  PR[GP1:91,1] = PR[GP1:90,1] + 27.012;
   1:  PR[GP1:91,2] = PR[GP1:90,2] + -31.910;
   1:L PR[91] R[100]mm/sec CNT100;
   1:  PR[GP1:91,1] = PR[GP1:90,1] + 36.564;
   1:  PR[GP1:91,2] = PR[GP1:90,2] + -34.385;
   1:L PR[91] R[100]mm/sec CNT100;
   1:  PR[GP1:91,1] = PR[GP1:90,1] + 37.852;
   1:  PR[GP1:91,2] = PR[GP1:90,2] + -34.408;
   1:L PR[91] R[100]mm/sec CNT100;
   1:  PR[GP1:91,1] = PR[GP1:90,1] + 46.562;
   1:  PR[GP1:91,2] = PR[GP1:90,2] + -33.753;
   1:L PR[91] R[100]mm/sec CNT100;
   1:  PR[GP1:91,1] = PR[GP1:90,1] + 48.244;
   1:  PR[GP1:91,2] = PR[GP1:90,2] + -33.466;
   1:L PR[91] R[100]mm/sec CNT100;
   1:  PR[GP1:91,1] = PR[GP1:90,1] + 49.855;
   1:  PR[GP1:91,2] = PR[GP1:90,2] + -32.868;
   1:L PR[91] R[100]mm/sec CNT100;
   1:  PR[GP1:91,1] = PR[GP1:90,1] + 57.348;
   1:  PR[GP1:91,2] = PR[GP1:90,2] + -29.641;
   1:L PR[91] R[100]mm/sec CNT100;
   1:  PR[GP1:91,1] = PR[GP1:90,1] + 59.071;
   1:  PR[GP1:91,2] = PR[GP1:90,2] + -28.602;
   1:L PR[91] R[100]mm/sec CNT100;
   1:  PR[GP1:91,1] = PR[GP1:90,1] + 60.599;
   1:  PR[GP1:91,2] = PR[GP1:90,2] + -27.235;
   1:L PR[91] R[100]mm/sec CNT100;
   1:  PR[GP1:91,1] = PR[GP1:90,1] + 66.288;
   1:  PR[GP1:91,2] = PR[GP1:90,2] + -22.049;
   1:L PR[91] R[100]mm/sec CNT100;
   1:  PR[GP1:91,1] = PR[GP1:90,1] + 67.643;
   1:  PR[GP1:91,2] = PR[GP1:90,2] + -20.283;
   1:L PR[91] R[100]mm/sec CNT100;
   1:  PR[GP1:91,1] = PR[GP1:90,1] + 68.674;
   1:  PR[GP1:91,2] = PR[GP1:90,2] + -18.240;
   1:L PR[91] R[100]mm/sec CNT100;
   1:  PR[GP1:91,1] = PR[GP1:90,1] + 72.196;
   1:  PR[GP1:91,2] = PR[GP1:90,2] + -11.780;
   1:L PR[91] R[100]mm/sec CNT100;
   1:  PR[GP1:91,1] = PR[GP1:90,1] + 72.845;
   1:  PR[GP1:91,2] = PR[GP1:90,2] + -9.525;
   1:L PR[91] R[100]mm/sec CNT100;
   1:  PR[GP1:91,1] = PR[GP1:90,1] + 73.072;
   1:  PR[GP1:91,2] = PR[GP1:90,2] + -7.101;
   1:L PR[91] R[100]mm/sec CNT100;
   1:  PR[GP1:91,1] = PR[GP1:90,1] + 74.248;
   1:  PR[GP1:91,2] = PR[GP1:90,2] + -0.050;
   1:L PR[91] R[100]mm/sec CNT100;
   1:  PR[GP1:91,1] = PR[GP1:90,1] + 74.013;
   1:  PR[GP1:91,2] = PR[GP1:90,2] + 2.454;
   1:L PR[91] R[100]mm/sec CNT100;
   1:  PR[GP1:91,1] = PR[GP1:90,1] + 72.851;
   1:  PR[GP1:91,2] = PR[GP1:90,2] + 9.360;
   1:L PR[91] R[100]mm/sec CNT100;
   1:  PR[GP1:91,1] = PR[GP1:90,1] + 72.193;
   1:  PR[GP1:91,2] = PR[GP1:90,2] + 11.646;
   1:L PR[91] R[100]mm/sec CNT100;
   1:  PR[GP1:91,1] = PR[GP1:90,1] + 71.110;
   1:  PR[GP1:91,2] = PR[GP1:90,2] + 13.791;
   1:L PR[91] R[100]mm/sec CNT100;
   1:  PR[GP1:91,1] = PR[GP1:90,1] + 67.649;
   1:  PR[GP1:91,2] = PR[GP1:90,2] + 20.132;
   1:L PR[91] R[100]mm/sec CNT100;
   1:  PR[GP1:91,1] = PR[GP1:90,1] + 66.290;
   1:  PR[GP1:91,2] = PR[GP1:90,2] + 21.903;
   1:L PR[91] R[100]mm/sec CNT100;
   1:  PR[GP1:91,1] = PR[GP1:90,1] + 64.589;
   1:  PR[GP1:91,2] = PR[GP1:90,2] + 23.424;
   1:L PR[91] R[100]mm/sec CNT100;
   1:  PR[GP1:91,1] = PR[GP1:90,1] + 59.068;
   1:  PR[GP1:91,2] = PR[GP1:90,2] + 28.459;
   1:L PR[91] R[100]mm/sec CNT100;
   1:  PR[GP1:91,1] = PR[GP1:90,1] + 57.361;
   1:  PR[GP1:91,2] = PR[GP1:90,2] + 29.489;
   1:L PR[91] R[100]mm/sec CNT100;
   1:  PR[GP1:91,1] = PR[GP1:90,1] + 55.422;
   1:  PR[GP1:91,2] = PR[GP1:90,2] + 30.209;
   1:L PR[91] R[100]mm/sec CNT100;
   1:  PR[GP1:91,1] = PR[GP1:90,1] + 48.228;
   1:  PR[GP1:91,2] = PR[GP1:90,2] + 33.325;
   1:L PR[91] R[100]mm/sec CNT100;
   1:  PR[GP1:91,1] = PR[GP1:90,1] + 46.562;
   1:  PR[GP1:91,2] = PR[GP1:90,2] + 33.609;
   1:L PR[91] R[100]mm/sec CNT100;
   1:  PR[GP1:91,1] = PR[GP1:90,1] + 37.852;
   1:  PR[GP1:91,2] = PR[GP1:90,2] + 34.264;
   1:L PR[91] R[100]mm/sec CNT100;
   1:  PR[GP1:91,1] = PR[GP1:90,1] + 36.550;
   1:  PR[GP1:91,2] = PR[GP1:90,2] + 34.240;
   1:L PR[91] R[100]mm/sec CNT100;
   1:  PR[GP1:91,1] = PR[GP1:90,1] + 35.262;
   1:  PR[GP1:91,2] = PR[GP1:90,2] + 33.973;
   1:L PR[91] R[100]mm/sec CNT100;
   1:  PR[GP1:91,1] = PR[GP1:90,1] + 26.164;
   1:  PR[GP1:91,2] = PR[GP1:90,2] + 31.593;
   1:L PR[91] R[100]mm/sec CNT100;
   1:  PR[GP1:91,1] = PR[GP1:90,1] + 25.404;
   1:  PR[GP1:91,2] = PR[GP1:90,2] + 31.278;
   1:L PR[91] R[100]mm/sec CNT100;
   1:  PR[GP1:91,1] = PR[GP1:90,1] + 16.243;
   1:  PR[GP1:91,2] = PR[GP1:90,2] + 25.205;
   1:L PR[91] R[100]mm/sec CNT100;
   1:  PR[GP1:91,1] = PR[GP1:90,1] + 15.999;
   1:  PR[GP1:91,2] = PR[GP1:90,2] + 24.970;
   1:L PR[91] R[100]mm/sec CNT100;
   1:  PR[GP1:91,1] = PR[GP1:90,1] + 15.765;
   1:  PR[GP1:91,2] = PR[GP1:90,2] + 24.641;
   1:L PR[91] R[100]mm/sec CNT100;
   1:  PR[GP1:91,1] = PR[GP1:90,1] + 9.192;
   1:  PR[GP1:91,2] = PR[GP1:90,2] + 16.055;
   1:L PR[91] R[100]mm/sec CNT100;
   1:  PR[GP1:91,1] = PR[GP1:90,1] + 5.551;
   1:  PR[GP1:91,2] = PR[GP1:90,2] + 5.303;
   1:L PR[91] R[100]mm/sec CNT100;
   1:  PR[GP1:91,1] = PR[GP1:90,1] + 5.269;
   1:  PR[GP1:91,2] = PR[GP1:90,2] + 4.511;
   1:L PR[91] R[100]mm/sec CNT100;
   1:  PR[GP1:91,1] = PR[GP1:90,1] + 4.562;
   1:  PR[GP1:91,2] = PR[GP1:90,2] + 2.847;
   1:L PR[91] R[100]mm/sec CNT100;
   1:  PR[GP1:91,1] = PR[GP1:90,1] + 4.109;
   1:  PR[GP1:91,2] = PR[GP1:90,2] + 2.447;
   1:L PR[91] R[100]mm/sec CNT100;
   1:  PR[GP1:91,1] = PR[GP1:90,1] + 3.490;
   1:  PR[GP1:91,2] = PR[GP1:90,2] + 1.809;
   1:L PR[91] R[100]mm/sec CNT100;
   1:  PR[GP1:91,1] = PR[GP1:90,1] + 2.541;
   1:  PR[GP1:91,2] = PR[GP1:90,2] + 1.338;
   1:L PR[91] R[100]mm/sec CNT100;
   1:  PR[GP1:91,1] = PR[GP1:90,1] + 1.710;
   1:  PR[GP1:91,2] = PR[GP1:90,2] + 0.866;
   1:L PR[91] R[100]mm/sec CNT100;
   1:  PR[GP1:91,1] = PR[GP1:90,1] + 0.434;
   1:  PR[GP1:91,2] = PR[GP1:90,2] + 0.582;
   1:L PR[91] R[100]mm/sec CNT100;
   1:  PR[GP1:91,1] = PR[GP1:90,1] + 0.167;
   1:  PR[GP1:91,2] = PR[GP1:90,2] + 0.581;
   1:L PR[91] R[100]mm/sec CNT100;
   1:  ! -- Layer/Ebene 26 -- !;
   1:  PR[91] = PR[90];
   1:  PR[GP1:91,1] = PR[GP1:90,1] + -3.038;
   1:  PR[GP1:91,2] = PR[GP1:90,2] + 1.930;
   1:  PR[GP1:91,3] = PR[GP1:90,3] + 16.165;
   1:L PR[91] R[100]mm/sec CNT100;
   1:  PR[GP1:91,1] = PR[GP1:90,1] + -3.247;
   1:  PR[GP1:91,2] = PR[GP1:90,2] + 2.101;
   1:L PR[91] R[100]mm/sec CNT100;
   1:  PR[GP1:91,1] = PR[GP1:90,1] + -5.297;
   1:  PR[GP1:91,2] = PR[GP1:90,2] + 5.692;
   1:L PR[91] R[100]mm/sec CNT100;
   1:  PR[GP1:91,1] = PR[GP1:90,1] + -8.666;
   1:  PR[GP1:91,2] = PR[GP1:90,2] + 15.614;
   1:L PR[91] R[100]mm/sec CNT100;
   1:  PR[GP1:91,1] = PR[GP1:90,1] + -9.016;
   1:  PR[GP1:91,2] = PR[GP1:90,2] + 16.315;
   1:L PR[91] R[100]mm/sec CNT100;
   1:  PR[GP1:91,1] = PR[GP1:90,1] + -15.863;
   1:  PR[GP1:91,2] = PR[GP1:90,2] + 25.105;
   1:L PR[91] R[100]mm/sec CNT100;
   1:  PR[GP1:91,1] = PR[GP1:90,1] + -15.871;
   1:  PR[GP1:91,2] = PR[GP1:90,2] + 25.113;
   1:L PR[91] R[100]mm/sec CNT100;
   1:  PR[GP1:91,1] = PR[GP1:90,1] + -16.894;
   1:  PR[GP1:91,2] = PR[GP1:90,2] + 25.777;
   1:L PR[91] R[100]mm/sec CNT100;
   1:  PR[GP1:91,1] = PR[GP1:90,1] + -25.306;
   1:  PR[GP1:91,2] = PR[GP1:90,2] + 31.357;
   1:L PR[91] R[100]mm/sec CNT100;
   1:  PR[GP1:91,1] = PR[GP1:90,1] + -25.616;
   1:  PR[GP1:91,2] = PR[GP1:90,2] + 31.486;
   1:L PR[91] R[100]mm/sec CNT100;
   1:  PR[GP1:91,1] = PR[GP1:90,1] + -26.016;
   1:  PR[GP1:91,2] = PR[GP1:90,2] + 31.569;
   1:L PR[91] R[100]mm/sec CNT100;
   1:  PR[GP1:91,1] = PR[GP1:90,1] + -36.376;
   1:  PR[GP1:91,2] = PR[GP1:90,2] + 34.252;
   1:L PR[91] R[100]mm/sec CNT100;
   1:  PR[GP1:91,1] = PR[GP1:90,1] + -37.230;
   1:  PR[GP1:91,2] = PR[GP1:90,2] + 34.267;
   1:L PR[91] R[100]mm/sec CNT100;
   1:  PR[GP1:91,1] = PR[GP1:90,1] + -46.678;
   1:  PR[GP1:91,2] = PR[GP1:90,2] + 33.556;
   1:L PR[91] R[100]mm/sec CNT100;
   1:  PR[GP1:91,1] = PR[GP1:90,1] + -47.966;
   1:  PR[GP1:91,2] = PR[GP1:90,2] + 33.337;
   1:L PR[91] R[100]mm/sec CNT100;
   1:  PR[GP1:91,1] = PR[GP1:90,1] + -49.203;
   1:  PR[GP1:91,2] = PR[GP1:90,2] + 32.877;
   1:L PR[91] R[100]mm/sec CNT100;
   1:  PR[GP1:91,1] = PR[GP1:90,1] + -57.331;
   1:  PR[GP1:91,2] = PR[GP1:90,2] + 29.376;
   1:L PR[91] R[100]mm/sec CNT100;
   1:  PR[GP1:91,1] = PR[GP1:90,1] + -58.735;
   1:  PR[GP1:91,2] = PR[GP1:90,2] + 28.529;
   1:L PR[91] R[100]mm/sec CNT100;
   1:  PR[GP1:91,1] = PR[GP1:90,1] + -59.985;
   1:  PR[GP1:91,2] = PR[GP1:90,2] + 27.411;
   1:L PR[91] R[100]mm/sec CNT100;
   1:  PR[GP1:91,1] = PR[GP1:90,1] + -66.157;
   1:  PR[GP1:91,2] = PR[GP1:90,2] + 21.787;
   1:L PR[91] R[100]mm/sec CNT100;
   1:  PR[GP1:91,1] = PR[GP1:90,1] + -67.296;
   1:  PR[GP1:91,2] = PR[GP1:90,2] + 20.302;
   1:L PR[91] R[100]mm/sec CNT100;
   1:  PR[GP1:91,1] = PR[GP1:90,1] + -68.168;
   1:  PR[GP1:91,2] = PR[GP1:90,2] + 18.574;
   1:L PR[91] R[100]mm/sec CNT100;
   1:  PR[GP1:91,1] = PR[GP1:90,1] + -71.988;
   1:  PR[GP1:91,2] = PR[GP1:90,2] + 11.562;
   1:L PR[91] R[100]mm/sec CNT100;
   1:  PR[GP1:91,1] = PR[GP1:90,1] + -72.543;
   1:  PR[GP1:91,2] = PR[GP1:90,2] + 9.635;
   1:L PR[91] R[100]mm/sec CNT100;
   1:  PR[GP1:91,1] = PR[GP1:90,1] + -72.738;
   1:  PR[GP1:91,2] = PR[GP1:90,2] + 7.551;
   1:L PR[91] R[100]mm/sec CNT100;
   1:  PR[GP1:91,1] = PR[GP1:90,1] + -74.013;
   1:  PR[GP1:91,2] = PR[GP1:90,2] + -0.094;
   1:L PR[91] R[100]mm/sec CNT100;
   1:  PR[GP1:91,1] = PR[GP1:90,1] + -73.809;
   1:  PR[GP1:91,2] = PR[GP1:90,2] + -2.269;
   1:L PR[91] R[100]mm/sec CNT100;
   1:  PR[GP1:91,1] = PR[GP1:90,1] + -72.549;
   1:  PR[GP1:91,2] = PR[GP1:90,2] + -9.758;
   1:L PR[91] R[100]mm/sec CNT100;
   1:  PR[GP1:91,1] = PR[GP1:90,1] + -71.985;
   1:  PR[GP1:91,2] = PR[GP1:90,2] + -11.715;
   1:L PR[91] R[100]mm/sec CNT100;
   1:  PR[GP1:91,1] = PR[GP1:90,1] + -71.056;
   1:  PR[GP1:91,2] = PR[GP1:90,2] + -13.556;
   1:L PR[91] R[100]mm/sec CNT100;
   1:  PR[GP1:91,1] = PR[GP1:90,1] + -67.302;
   1:  PR[GP1:91,2] = PR[GP1:90,2] + -20.438;
   1:L PR[91] R[100]mm/sec CNT100;
   1:  PR[GP1:91,1] = PR[GP1:90,1] + -66.158;
   1:  PR[GP1:91,2] = PR[GP1:90,2] + -21.929;
   1:L PR[91] R[100]mm/sec CNT100;
   1:  PR[GP1:91,1] = PR[GP1:90,1] + -64.721;
   1:  PR[GP1:91,2] = PR[GP1:90,2] + -23.215;
   1:L PR[91] R[100]mm/sec CNT100;
   1:  PR[GP1:91,1] = PR[GP1:90,1] + -58.732;
   1:  PR[GP1:91,2] = PR[GP1:90,2] + -28.674;
   1:L PR[91] R[100]mm/sec CNT100;
   1:  PR[GP1:91,1] = PR[GP1:90,1] + -57.344;
   1:  PR[GP1:91,2] = PR[GP1:90,2] + -29.512;
   1:L PR[91] R[100]mm/sec CNT100;
   1:  PR[GP1:91,1] = PR[GP1:90,1] + -55.754;
   1:  PR[GP1:91,2] = PR[GP1:90,2] + -30.102;
   1:L PR[91] R[100]mm/sec CNT100;
   1:  PR[GP1:91,1] = PR[GP1:90,1] + -47.950;
   1:  PR[GP1:91,2] = PR[GP1:90,2] + -33.483;
   1:L PR[91] R[100]mm/sec CNT100;
   1:  PR[GP1:91,1] = PR[GP1:90,1] + -46.678;
   1:  PR[GP1:91,2] = PR[GP1:90,2] + -33.700;
   1:L PR[91] R[100]mm/sec CNT100;
   1:  PR[GP1:91,1] = PR[GP1:90,1] + -37.230;
   1:  PR[GP1:91,2] = PR[GP1:90,2] + -34.411;
   1:L PR[91] R[100]mm/sec CNT100;
   1:  PR[GP1:91,1] = PR[GP1:90,1] + -36.361;
   1:  PR[GP1:91,2] = PR[GP1:90,2] + -34.395;
   1:L PR[91] R[100]mm/sec CNT100;
   1:  PR[GP1:91,1] = PR[GP1:90,1] + -35.498;
   1:  PR[GP1:91,2] = PR[GP1:90,2] + -34.216;
   1:L PR[91] R[100]mm/sec CNT100;
   1:  PR[GP1:91,1] = PR[GP1:90,1] + -25.630;
   1:  PR[GP1:91,2] = PR[GP1:90,2] + -31.635;
   1:L PR[91] R[100]mm/sec CNT100;
   1:  PR[GP1:91,1] = PR[GP1:90,1] + -25.306;
   1:  PR[GP1:91,2] = PR[GP1:90,2] + -31.501;
   1:L PR[91] R[100]mm/sec CNT100;
   1:  PR[GP1:91,1] = PR[GP1:90,1] + -16.893;
   1:  PR[GP1:91,2] = PR[GP1:90,2] + -25.921;
   1:L PR[91] R[100]mm/sec CNT100;
   1:  PR[GP1:91,1] = PR[GP1:90,1] + -15.871;
   1:  PR[GP1:91,2] = PR[GP1:90,2] + -25.257;
   1:L PR[91] R[100]mm/sec CNT100;
   1:  PR[GP1:91,1] = PR[GP1:90,1] + -15.863;
   1:  PR[GP1:91,2] = PR[GP1:90,2] + -25.249;
   1:L PR[91] R[100]mm/sec CNT100;
   1:  PR[GP1:91,1] = PR[GP1:90,1] + -9.016;
   1:  PR[GP1:91,2] = PR[GP1:90,2] + -16.459;
   1:L PR[91] R[100]mm/sec CNT100;
   1:  PR[GP1:91,1] = PR[GP1:90,1] + -8.666;
   1:  PR[GP1:91,2] = PR[GP1:90,2] + -15.760;
   1:L PR[91] R[100]mm/sec CNT100;
   1:  PR[GP1:91,1] = PR[GP1:90,1] + -5.314;
   1:  PR[GP1:91,2] = PR[GP1:90,2] + -5.886;
   1:L PR[91] R[100]mm/sec CNT100;
   1:  PR[GP1:91,1] = PR[GP1:90,1] + -4.646;
   1:  PR[GP1:91,2] = PR[GP1:90,2] + -4.012;
   1:L PR[91] R[100]mm/sec CNT100;
   1:  PR[GP1:91,1] = PR[GP1:90,1] + -4.343;
   1:  PR[GP1:91,2] = PR[GP1:90,2] + -3.300;
   1:L PR[91] R[100]mm/sec CNT100;
   1:  PR[GP1:91,1] = PR[GP1:90,1] + -3.459;
   1:  PR[GP1:91,2] = PR[GP1:90,2] + -2.521;
   1:L PR[91] R[100]mm/sec CNT100;
   1:  PR[GP1:91,1] = PR[GP1:90,1] + -3.000;
   1:  PR[GP1:91,2] = PR[GP1:90,2] + -2.048;
   1:L PR[91] R[100]mm/sec CNT100;
   1:  PR[GP1:91,1] = PR[GP1:90,1] + -2.698;
   1:  PR[GP1:91,2] = PR[GP1:90,2] + -1.927;
   1:L PR[91] R[100]mm/sec CNT100;
   1:  PR[GP1:91,1] = PR[GP1:90,1] + -1.175;
   1:  PR[GP1:91,2] = PR[GP1:90,2] + -1.151;
   1:L PR[91] R[100]mm/sec CNT100;
   1:  PR[GP1:91,1] = PR[GP1:90,1] + -0.862;
   1:  PR[GP1:91,2] = PR[GP1:90,2] + -0.973;
   1:L PR[91] R[100]mm/sec CNT100;
   1:  PR[GP1:91,1] = PR[GP1:90,1] + -0.218;
   1:  PR[GP1:91,2] = PR[GP1:90,2] + -0.841;
   1:L PR[91] R[100]mm/sec CNT100;
   1:  PR[GP1:91,1] = PR[GP1:90,1] + 3.251;
   1:  PR[GP1:91,2] = PR[GP1:90,2] + -2.074;
   1:L PR[91] R[100]mm/sec CNT100;
   1:  PR[GP1:91,1] = PR[GP1:90,1] + 3.461;
   1:  PR[GP1:91,2] = PR[GP1:90,2] + -2.246;
   1:L PR[91] R[100]mm/sec CNT100;
   1:  PR[GP1:91,1] = PR[GP1:90,1] + 4.422;
   1:  PR[GP1:91,2] = PR[GP1:90,2] + -3.937;
   1:L PR[91] R[100]mm/sec CNT100;
   1:  PR[GP1:91,1] = PR[GP1:90,1] + 5.233;
   1:  PR[GP1:91,2] = PR[GP1:90,2] + -5.481;
   1:L PR[91] R[100]mm/sec CNT100;
   1:  PR[GP1:91,1] = PR[GP1:90,1] + 5.490;
   1:  PR[GP1:91,2] = PR[GP1:90,2] + -5.781;
   1:L PR[91] R[100]mm/sec CNT100;
   1:  PR[GP1:91,1] = PR[GP1:90,1] + 8.877;
   1:  PR[GP1:91,2] = PR[GP1:90,2] + -15.755;
   1:L PR[91] R[100]mm/sec CNT100;
   1:  PR[GP1:91,1] = PR[GP1:90,1] + 9.227;
   1:  PR[GP1:91,2] = PR[GP1:90,2] + -16.453;
   1:L PR[91] R[100]mm/sec CNT100;
   1:  PR[GP1:91,1] = PR[GP1:90,1] + 16.074;
   1:  PR[GP1:91,2] = PR[GP1:90,2] + -25.248;
   1:L PR[91] R[100]mm/sec CNT100;
   1:  PR[GP1:91,1] = PR[GP1:90,1] + 16.082;
   1:  PR[GP1:91,2] = PR[GP1:90,2] + -25.256;
   1:L PR[91] R[100]mm/sec CNT100;
   1:  PR[GP1:91,1] = PR[GP1:90,1] + 17.106;
   1:  PR[GP1:91,2] = PR[GP1:90,2] + -25.921;
   1:L PR[91] R[100]mm/sec CNT100;
   1:  PR[GP1:91,1] = PR[GP1:90,1] + 25.517;
   1:  PR[GP1:91,2] = PR[GP1:90,2] + -31.500;
   1:L PR[91] R[100]mm/sec CNT100;
   1:  PR[GP1:91,1] = PR[GP1:90,1] + 25.827;
   1:  PR[GP1:91,2] = PR[GP1:90,2] + -31.628;
   1:L PR[91] R[100]mm/sec CNT100;
   1:  PR[GP1:91,1] = PR[GP1:90,1] + 26.227;
   1:  PR[GP1:91,2] = PR[GP1:90,2] + -31.712;
   1:L PR[91] R[100]mm/sec CNT100;
   1:  PR[GP1:91,1] = PR[GP1:90,1] + 36.588;
   1:  PR[GP1:91,2] = PR[GP1:90,2] + -34.396;
   1:L PR[91] R[100]mm/sec CNT100;
   1:  PR[GP1:91,1] = PR[GP1:90,1] + 37.442;
   1:  PR[GP1:91,2] = PR[GP1:90,2] + -34.411;
   1:L PR[91] R[100]mm/sec CNT100;
   1:  PR[GP1:91,1] = PR[GP1:90,1] + 46.890;
   1:  PR[GP1:91,2] = PR[GP1:90,2] + -33.700;
   1:L PR[91] R[100]mm/sec CNT100;
   1:  PR[GP1:91,1] = PR[GP1:90,1] + 48.178;
   1:  PR[GP1:91,2] = PR[GP1:90,2] + -33.481;
   1:L PR[91] R[100]mm/sec CNT100;
   1:  PR[GP1:91,1] = PR[GP1:90,1] + 49.415;
   1:  PR[GP1:91,2] = PR[GP1:90,2] + -33.021;
   1:L PR[91] R[100]mm/sec CNT100;
   1:  PR[GP1:91,1] = PR[GP1:90,1] + 57.543;
   1:  PR[GP1:91,2] = PR[GP1:90,2] + -29.521;
   1:L PR[91] R[100]mm/sec CNT100;
   1:  PR[GP1:91,1] = PR[GP1:90,1] + 58.947;
   1:  PR[GP1:91,2] = PR[GP1:90,2] + -28.674;
   1:L PR[91] R[100]mm/sec CNT100;
   1:  PR[GP1:91,1] = PR[GP1:90,1] + 60.198;
   1:  PR[GP1:91,2] = PR[GP1:90,2] + -27.556;
   1:L PR[91] R[100]mm/sec CNT100;
   1:  PR[GP1:91,1] = PR[GP1:90,1] + 66.369;
   1:  PR[GP1:91,2] = PR[GP1:90,2] + -21.930;
   1:L PR[91] R[100]mm/sec CNT100;
   1:  PR[GP1:91,1] = PR[GP1:90,1] + 67.509;
   1:  PR[GP1:91,2] = PR[GP1:90,2] + -20.444;
   1:L PR[91] R[100]mm/sec CNT100;
   1:  PR[GP1:91,1] = PR[GP1:90,1] + 68.381;
   1:  PR[GP1:91,2] = PR[GP1:90,2] + -18.717;
   1:L PR[91] R[100]mm/sec CNT100;
   1:  PR[GP1:91,1] = PR[GP1:90,1] + 72.201;
   1:  PR[GP1:91,2] = PR[GP1:90,2] + -11.709;
   1:L PR[91] R[100]mm/sec CNT100;
   1:  PR[GP1:91,1] = PR[GP1:90,1] + 72.756;
   1:  PR[GP1:91,2] = PR[GP1:90,2] + -9.782;
   1:L PR[91] R[100]mm/sec CNT100;
   1:  PR[GP1:91,1] = PR[GP1:90,1] + 72.951;
   1:  PR[GP1:91,2] = PR[GP1:90,2] + -7.699;
   1:L PR[91] R[100]mm/sec CNT100;
   1:  PR[GP1:91,1] = PR[GP1:90,1] + 74.227;
   1:  PR[GP1:91,2] = PR[GP1:90,2] + -0.050;
   1:L PR[91] R[100]mm/sec CNT100;
   1:  PR[GP1:91,1] = PR[GP1:90,1] + 74.023;
   1:  PR[GP1:91,2] = PR[GP1:90,2] + 2.126;
   1:L PR[91] R[100]mm/sec CNT100;
   1:  PR[GP1:91,1] = PR[GP1:90,1] + 72.762;
   1:  PR[GP1:91,2] = PR[GP1:90,2] + 9.617;
   1:L PR[91] R[100]mm/sec CNT100;
   1:  PR[GP1:91,1] = PR[GP1:90,1] + 72.198;
   1:  PR[GP1:91,2] = PR[GP1:90,2] + 11.575;
   1:L PR[91] R[100]mm/sec CNT100;
   1:  PR[GP1:91,1] = PR[GP1:90,1] + 71.270;
   1:  PR[GP1:91,2] = PR[GP1:90,2] + 13.415;
   1:L PR[91] R[100]mm/sec CNT100;
   1:  PR[GP1:91,1] = PR[GP1:90,1] + 67.515;
   1:  PR[GP1:91,2] = PR[GP1:90,2] + 20.293;
   1:L PR[91] R[100]mm/sec CNT100;
   1:  PR[GP1:91,1] = PR[GP1:90,1] + 66.371;
   1:  PR[GP1:91,2] = PR[GP1:90,2] + 21.784;
   1:L PR[91] R[100]mm/sec CNT100;
   1:  PR[GP1:91,1] = PR[GP1:90,1] + 64.933;
   1:  PR[GP1:91,2] = PR[GP1:90,2] + 23.070;
   1:L PR[91] R[100]mm/sec CNT100;
   1:  PR[GP1:91,1] = PR[GP1:90,1] + 58.945;
   1:  PR[GP1:91,2] = PR[GP1:90,2] + 28.532;
   1:L PR[91] R[100]mm/sec CNT100;
   1:  PR[GP1:91,1] = PR[GP1:90,1] + 57.557;
   1:  PR[GP1:91,2] = PR[GP1:90,2] + 29.369;
   1:L PR[91] R[100]mm/sec CNT100;
   1:  PR[GP1:91,1] = PR[GP1:90,1] + 55.966;
   1:  PR[GP1:91,2] = PR[GP1:90,2] + 29.960;
   1:L PR[91] R[100]mm/sec CNT100;
   1:  PR[GP1:91,1] = PR[GP1:90,1] + 48.162;
   1:  PR[GP1:91,2] = PR[GP1:90,2] + 33.339;
   1:L PR[91] R[100]mm/sec CNT100;
   1:  PR[GP1:91,1] = PR[GP1:90,1] + 46.890;
   1:  PR[GP1:91,2] = PR[GP1:90,2] + 33.556;
   1:L PR[91] R[100]mm/sec CNT100;
   1:  PR[GP1:91,1] = PR[GP1:90,1] + 37.442;
   1:  PR[GP1:91,2] = PR[GP1:90,2] + 34.267;
   1:L PR[91] R[100]mm/sec CNT100;
   1:  PR[GP1:91,1] = PR[GP1:90,1] + 36.573;
   1:  PR[GP1:91,2] = PR[GP1:90,2] + 34.251;
   1:L PR[91] R[100]mm/sec CNT100;
   1:  PR[GP1:91,1] = PR[GP1:90,1] + 35.710;
   1:  PR[GP1:91,2] = PR[GP1:90,2] + 34.072;
   1:L PR[91] R[100]mm/sec CNT100;
   1:  PR[GP1:91,1] = PR[GP1:90,1] + 25.841;
   1:  PR[GP1:91,2] = PR[GP1:90,2] + 31.490;
   1:L PR[91] R[100]mm/sec CNT100;
   1:  PR[GP1:91,1] = PR[GP1:90,1] + 25.517;
   1:  PR[GP1:91,2] = PR[GP1:90,2] + 31.356;
   1:L PR[91] R[100]mm/sec CNT100;
   1:  PR[GP1:91,1] = PR[GP1:90,1] + 17.107;
   1:  PR[GP1:91,2] = PR[GP1:90,2] + 25.777;
   1:L PR[91] R[100]mm/sec CNT100;
   1:  PR[GP1:91,1] = PR[GP1:90,1] + 16.082;
   1:  PR[GP1:91,2] = PR[GP1:90,2] + 25.112;
   1:L PR[91] R[100]mm/sec CNT100;
   1:  PR[GP1:91,1] = PR[GP1:90,1] + 16.074;
   1:  PR[GP1:91,2] = PR[GP1:90,2] + 25.104;
   1:L PR[91] R[100]mm/sec CNT100;
   1:  PR[GP1:91,1] = PR[GP1:90,1] + 9.227;
   1:  PR[GP1:91,2] = PR[GP1:90,2] + 16.309;
   1:L PR[91] R[100]mm/sec CNT100;
   1:  PR[GP1:91,1] = PR[GP1:90,1] + 8.877;
   1:  PR[GP1:91,2] = PR[GP1:90,2] + 15.609;
   1:L PR[91] R[100]mm/sec CNT100;
   1:  PR[GP1:91,1] = PR[GP1:90,1] + 5.526;
   1:  PR[GP1:91,2] = PR[GP1:90,2] + 5.742;
   1:L PR[91] R[100]mm/sec CNT100;
   1:  PR[GP1:91,1] = PR[GP1:90,1] + 4.859;
   1:  PR[GP1:91,2] = PR[GP1:90,2] + 3.870;
   1:L PR[91] R[100]mm/sec CNT100;
   1:  PR[GP1:91,1] = PR[GP1:90,1] + 4.556;
   1:  PR[GP1:91,2] = PR[GP1:90,2] + 3.156;
   1:L PR[91] R[100]mm/sec CNT100;
   1:  PR[GP1:91,1] = PR[GP1:90,1] + 3.672;
   1:  PR[GP1:91,2] = PR[GP1:90,2] + 2.378;
   1:L PR[91] R[100]mm/sec CNT100;
   1:  PR[GP1:91,1] = PR[GP1:90,1] + 3.213;
   1:  PR[GP1:91,2] = PR[GP1:90,2] + 1.905;
   1:L PR[91] R[100]mm/sec CNT100;
   1:  PR[GP1:91,1] = PR[GP1:90,1] + 2.912;
   1:  PR[GP1:91,2] = PR[GP1:90,2] + 1.783;
   1:L PR[91] R[100]mm/sec CNT100;
   1:  PR[GP1:91,1] = PR[GP1:90,1] + 1.388;
   1:  PR[GP1:91,2] = PR[GP1:90,2] + 1.007;
   1:L PR[91] R[100]mm/sec CNT100;
   1:  PR[GP1:91,1] = PR[GP1:90,1] + 1.075;
   1:  PR[GP1:91,2] = PR[GP1:90,2] + 0.829;
   1:L PR[91] R[100]mm/sec CNT100;
   1:  PR[GP1:91,1] = PR[GP1:90,1] + 0.431;
   1:  PR[GP1:91,2] = PR[GP1:90,2] + 0.697;
   1:L PR[91] R[100]mm/sec CNT100 TB   .50sec,CALL END_PUD;
   1:  DO[117:Laser Start]=OFF;
   1:  !Sicherheitspunkt!;
   1:  PR[92] = PR[91];
   1:  PR[92] = PR[GP1:92,3] + 50;
   1:J PR[92];
   1:  WAIT   5.00(sec);
   1:  DO[119:Gas]=OFF;
   1:  CALL HOME_ALL;
/POS
/END
